// TIA Portal project "MEC10112tHiL2019" (V15)

(* hardware
DEVICE "S7-1200 station_1"  S7-1200 Station
   slot 0: "Rack_0"  S7-1200 Rack  Rack  V1.0
   slot 1: "Simulated Plant Process"  CPU 1214C DC/DC/DC  6ES7 214-1AG40-0XB0  V4.2
      slot 3: "AQ 1x12BIT_1"  AQ1 signal board  6ES7 232-4HA30-0XB0  V1.0
DEVICE "HMI_1"  KTP700 Basic PN
   slot 0: "HMI_1"  KTP700 Basic PN  6AV2 123-2GB03-0AX0  15.0.0.0
   slot 1: "HMI_RT_1"  KTP700 Basic PN  6AV2 123-2GB03-0AX0  15.0.0.0
   slot 5: "HMI_1.IE_CP_1"  PROFINET Interface  15.0.0.0
      slot 1: "PROFINET Interface_1"  PROFINET Interface
         slot 1: "Port_1"  Port
DEVICE "S7-1200 station_2"  S7-1200 Station
   slot 0: "Rack_0"  S7-1200 Rack  Rack  V1.0
   slot 1: "Control Panel PLC"  CPU 1214C AC/DC/Rly  6ES7 214-1BG31-0XB0  V3.0
   slot 3: "AQ 1x12BIT_1"  AQ1 signal board  6ES7 232-4HA30-0XB0  V1.0
DEVICE "SCADA_Display"  SIMATIC PC station
   slot 0: "SIMATIC PC station"  Rail  SIMATIC PC-Station  V1.0
      slot 125: "Stationmanager"  Station_Manager  V6.0.4
   slot 1: "HMI_RT_2"  WinCC RT Advanced  6AV2 104-0xxxx-xxxx  15.0.0.0
      slot 33792: "Host interface"  Host interface
   slot 2: "IE general_1"  IE General  IE_CP  V8.2.0
*)

// ===== PLC "Simulated Plant Process"  CPU 1214C DC/DC/DC =====

VAR_GLOBAL   // PLC tag table "Default tag table"
   "Level" AT %QW80 : Int;
   "OpenV101" AT %I0.0 : Bool;
   "OpenV102" AT %I0.1 : Bool;
   "OpenV103" AT %I0.2 : Bool;
   "OpenV104" AT %I0.3 : Bool;
   "V101OpenLSW" AT %Q0.0 : Bool;
   "V101CloseLSW" AT %Q0.1 : Bool;
   "V102OpenLSW" AT %Q0.2 : Bool;
   "V102CloseLSW" AT %Q0.3 : Bool;
   "V103OpenLSW" AT %Q0.4 : Bool;
   "V103CloseLSW" AT %Q0.5 : Bool;
   "V104OpenLSW" AT %Q0.6 : Bool;
   "V104CloseLSW" AT %Q0.7 : Bool;
   "RunMix" AT %I0.4 : Bool;
   "MinimumHeatTankLevel" AT %Q1.0 : Bool;   // Liquid Level Reached in heating tank
   "MixerRunning" AT %Q1.4 : Bool;
   "Prod_A_Available" AT %Q1.2 : Bool;
   "Prod_B_Available" AT %Q1.3 : Bool;
   "Bottle_Sim_output" AT %Q1.1 : Bool;   // Added output to simulate bottle presence
END_VAR

DATA_BLOCK "TankLevel"   // DB1
{ S7_Optimized_Access := 'FALSE' }
VERSION : 0.1
// stored: InstanceOfName AnalogueOutput_type1
"AnalogueOutput_type1"
BEGIN
END_DATA_BLOCK

DATA_BLOCK "V101"   // DB2
{ S7_Optimized_Access := 'TRUE' }
VERSION : 0.1
// stored: InstanceOfName ValveSim
"ValveSim"
BEGIN
END_DATA_BLOCK

DATA_BLOCK "V102"   // DB3
{ S7_Optimized_Access := 'TRUE' }
VERSION : 0.1
// stored: InstanceOfName ValveSim
"ValveSim"
BEGIN
END_DATA_BLOCK

DATA_BLOCK "V103"   // DB4
{ S7_Optimized_Access := 'TRUE' }
VERSION : 0.1
// stored: InstanceOfName ValveSim
"ValveSim"
BEGIN
END_DATA_BLOCK

DATA_BLOCK "V104"   // DB5
{ S7_Optimized_Access := 'TRUE' }
VERSION : 0.1
// stored: InstanceOfName ValveSim
"ValveSim"
BEGIN
END_DATA_BLOCK

DATA_BLOCK "TankSimulator_DB"   // DB6
{ S7_Optimized_Access := 'TRUE' }
VERSION : 0.1
// stored: InstanceOfName TankSimulator
"TankSimulator"
BEGIN
END_DATA_BLOCK

// folder: System blocks/Program resources

DATA_BLOCK "MixerFB"   // DB7
{ S7_Optimized_Access := 'TRUE' }
AUTHOR : Simatic
FAMILY : IEC
NAME : IEC_TMR
VERSION : 1.0
// stored: InstanceOfName IEC_TIMER
"IEC_TIMER"
BEGIN
END_DATA_BLOCK

// folder: (top level)

FUNCTION_BLOCK "AnalogueInput_type1"   // FB1, SCL
{ S7_Optimized_Access := 'FALSE' }
VERSION : 0.1
   VAR_INPUT
      ChannelAddress : Int;   // PLC Channel Address
      HR : Real := 100.0;   // High Range i.e. Maximum Value of Input Signal
      LR : Real;   // Low Range i.e. Minimum Value of Input Signal
      HSP : Real := 90.0;   // High Alarm Set Point Value
      LSP : Real := 10.0;   // Low Alarm Set Point value
      EnableHSP : Bool := true;   // Enable High Alarm
      EnableLSP : Bool := true;   // Enable Low Alarm
   END_VAR
   VAR_OUTPUT
      PV : Real;   // Process Variable (Scaled Value)
      HighAlarm : Bool;   // High Alarm HSP exceeded
      LowAlarm : Bool;   // Low Alarm LSP exceeded
      HighRangeError : Bool;   // A/D value Exceeds 27,648
      LowRangeError : Bool;   // A/D value lower than 0
   END_VAR
BEGIN
   //This Function Block reads in a value from an anaolgue input channel and
   //scales it between high range (HR) and a low range (LR) values.
   //It also sets high and low value alarms against high (HSP) and low (LSP) set points
   //If the value from the A/D converter exceeds either 0 or 27648 it also generates
   //range error bits

   #PV := ((INT_TO_REAL (#ChannelAddress)*(#HR - #LR))/ 27648.0) + #LR; // Read and scale A/D Value
   IF #EnableHSP=1 THEN                                                 // If High Alarm Enabled
       IF #PV > #HSP THEN                                               // Drive High Alarm
           #HighAlarm := 1;// Statement section IF
       ELSIF #PV< #HSP THEN
           #HighAlarm := 0;
       END_IF;  // Statement section IF
   END_IF;

   IF #EnableLSP=1 THEN                                               // If Low Alarm Enabled
       IF #PV< #LSP THEN                                              // Drive Low Alarm
           #LowAlarm := 1;// Statement section IF
       ELSIF #PV > #LSP THEN
           #LowAlarm := 0;
       END_IF;// Statement section IF
       ;
   END_IF;

   IF #ChannelAddress > 27648 THEN                                 // If A/D value Exceeds 27648
       #HighRangeError := 1;                                       //Out of high range error
       #PV := #HR;                                                 // Limit Output to maximum Value
   END_IF;
   IF #ChannelAddress < 0 THEN                                     // If A/D value is less than 0
       #LowRangeError := 1;                                        // Out of low range error
       #PV := #LR;                                                 // Limit Output to minimum value
   END_IF;
   IF (#ChannelAddress > 0) AND (#ChannelAddress < 27649) THEN     // if in range reset range errors
       #HighRangeError := 0;
       #LowRangeError := 0;
   END_IF;

   //Revision History
   //Tested 25/01/2016
   //Rev 1.0 Added range clipping and error bits
END_FUNCTION_BLOCK

FUNCTION_BLOCK "ValveSim"   // FB2, SCL
{ S7_Optimized_Access := 'TRUE' }
VERSION : 0.1
   VAR_INPUT
      OpenCMD : Bool;
      FaultEnable : Bool;
      OpTime : Int := 20;   // 100ms Increments
   END_VAR
   VAR_OUTPUT
      LimitOpenLSW : Bool;
      LimitCloseLSW : Bool;
   END_VAR
   VAR
      OpenTimer : DInt;
      CloseTimer : DInt;
   END_VAR
BEGIN
   // Valve Open Simulation
   IF #OpenCMD=1 THEN                      //Open CMD
       #OpenTimer := #OpenTimer + 1;       //Inrement Timer
       IF #OpenTimer>=#OpTime AND NOT #FaultEnable THEN   //If Timed value equals or exceeds operaton time
           #LimitOpenLSW := 1;             // Set Limit Switch Feedback
           #OpenTimer:=#OpTime;            // Limit Timer
       END_IF;
   ELSIF #OpenCMD=0 THEN                   // on Close command
       #OpenTimer := 0;                    // Reset Timer
       #LimitOpenLSW := 0;                 // Reset Limit Switch Feedback
   END_IF;

   // Valve Close Simulation
   IF #OpenCMD = 0 THEN                      //Close CMD
       #CloseTimer := #CloseTimer + 1;       //Inrement Timer
       IF #CloseTimer >= #OpTime THEN        //If Timed value equals or exceeds operaton time
           #LimitCloseLSW := 1;              // Set Limit Switch Feedback
           #CloseTimer := #OpTime;           // Limit Timer
       END_IF;
   ELSIF #OpenCMD = 1 THEN                  // on Open command
       #CloseTimer := 0;                    // Reset Timer
       #LimitCloseLSW := 0;                 // Reset Limit Switch Feedback
   END_IF;
END_FUNCTION_BLOCK

FUNCTION_BLOCK "TankSimulator"   // FB3, SCL
{ S7_Optimized_Access := 'TRUE' }
VERSION : 0.1
   VAR_INPUT
      InputValveA : Bool;
      InputValveB : Bool;
      OuputValve : Bool;
      DumpValve : Bool;
      RateA : Real := 0.1;   // litres per 0.1 s
      RateB : Real := 0.1;   // litres per 0.1 s
      RateOut : Real := 0.2;
      HeatLvl_SP : Real := 20.0;
      HR : Real := 110.0;
      LR : Real;
   END_VAR
   VAR_OUTPUT
      "Heat Level" : Bool;
      Level : Real;
   END_VAR
   VAR
      Delta : Real;   // Combined Level Increment
      SimLevel : Real;
   END_VAR
BEGIN
   // Mixing Tank Level Simulator
   // Called from Time Interupt 100mS
   // 
   // Level Change Calculation
   #Delta := 0;                // Reset Delta Change
   IF #InputValveA=1 THEN      // If input valve A open add its rate to Delta
       #Delta:=#Delta + #RateA;
   END_IF;
   IF #InputValveB=1 THEN      // If input valve B open add its rate to Delta
       #Delta := #Delta + #RateB;   
   END_IF;
   IF #OuputValve=1 THEN       // If Output valve open subtract its rate to Delta
       #Delta := #Delta - #RateOut;
   END_IF;
   IF #DumpValve=1 THEN    // If dump valve open level =0
       #Delta := 0;
       #SimLevel := 0;
   END_IF;

   #SimLevel := #SimLevel + #Delta;  // Level Summation
   IF #SimLevel>#HR THEN       // Limit Maximum Level
       #SimLevel := #HR;
   END_IF;
   IF #SimLevel<#LR THEN       // Limit Minimum Level
       #SimLevel := #LR;
   END_IF;

   // Level Above Heat Element
   IF #SimLevel>#HeatLvl_SP THEN // If level covers heating element
       #"Heat Level" := 1;
   ELSIF #SimLevel<#HeatLvl_SP THEN
       #"Heat Level" := 0;
   END_IF;

   // Output Level Simulation
   #Level := #SimLevel;
END_FUNCTION_BLOCK

FUNCTION_BLOCK "AnalogueOutput_type1"   // FB4, SCL
{ S7_Optimized_Access := 'FALSE' }
VERSION : 0.1
   VAR_INPUT
      OP : Real;   // Value to be output to D/A
      HR : Real := 100.0;   // Maximum Value of Output
      LR : Real;   // Minimum Value of Output
   END_VAR
   VAR_OUTPUT
      "Channel Address" : Int;   // D/A Channel Address
      HRexceeded : Bool;   // Input Signal Out of Upper Range
      LRexceeded : Bool;   // Input Signal Out of Lower Range
   END_VAR
BEGIN
   // Function Scales a Real Analogue Value to an integer
   // between 0 and 27648 for driving analogue output card
   // 
   IF (#LR < #OP) AND (#OP < #HR) THEN //If value within range reset error bits
       #HRexceeded := 0;
       #LRexceeded := 0;
   END_IF;
   //
   // Range Real Value
   #"Channel Address":= DINT_TO_INT(ROUND_DINT((#OP*27648.0)/(#HR-#LR)));
   //
   //Range Checking
   IF #OP > #HR THEN                   //Has value exceeded maximum value
       #"Channel Address" := 27648;    //Setoutput to maximum
       #HRexceeded := 1;               //Set error bit
   END_IF;
   IF #OP < #LR THEN                   //Has value exceeded minimum value
       #"Channel Address" := 0;        //Set output to minimum
       #LRexceeded := 1;               //Set error bit
   END_IF;

   //
   //Revision History
   //Rev 1.0 Added range clipping and range errors JMcW 26/01/2016
END_FUNCTION_BLOCK

ORGANIZATION_BLOCK "Main"   // OB1, LAD, ProgramCycle
TITLE = "Main Program Sweep (Cycle)"
{ S7_Optimized_Access := 'TRUE' }
VERSION : 0.1
   VAR_INPUT
      Initial_Call : Bool;   // Initial call of this OB
      Remanence : Bool;   // =True, if remanent data are available
   END_VAR
BEGIN

REGION Network 1: Simulated Tank Level Output Driver
   // Takes simulated value and creates a 0-10v analgue output
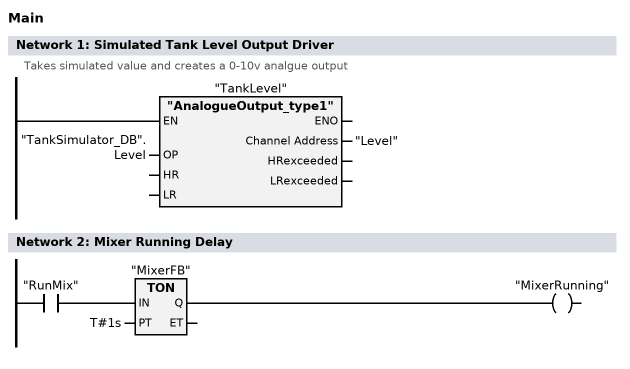
   RUNG wire#powerrail
      "TankLevel"(OP := "TankSimulator_DB".Level, HR :=, LR :=, "Channel Address" => "Level", HRexceeded =>, LRexceeded =>)
   END_RUNG
   // the same network as SCL:
   "TankLevel"(OP := "TankSimulator_DB".Level, "Channel Address" => "Level");   // "AnalogueOutput_type1"
END_REGION

REGION Network 2: Mixer Running Delay
   "MixerFB".TON(IN := "RunMix", PT := T#1s);
   "MixerRunning" := "MixerFB".Q;
END_REGION
END_ORGANIZATION_BLOCK

ORGANIZATION_BLOCK "Cyclic interrupt"   // OB30, LAD, CyclicInterrupt
TITLE = 100mS Cyclic Interupt
{ S7_Optimized_Access := 'TRUE' }
VERSION : 0.1
   VAR_INPUT
      Initial_Call : Bool;   // Initial call of this OB
      Event_Count : Int;   // Events discarded
   END_VAR
BEGIN

REGION Network 1: Inlet Valve 1 Simulation
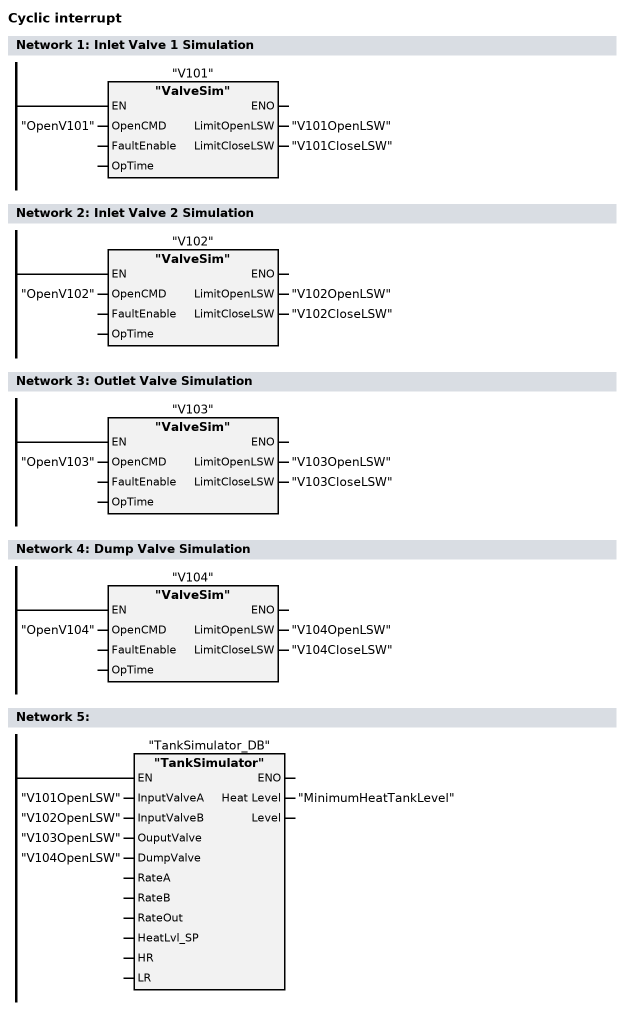
   RUNG wire#powerrail
      "V101"(OpenCMD := "OpenV101", FaultEnable :=, OpTime :=, LimitOpenLSW => "V101OpenLSW", LimitCloseLSW => "V101CloseLSW")
   END_RUNG
   // the same network as SCL:
   "V101"(OpenCMD := "OpenV101", LimitOpenLSW => "V101OpenLSW", LimitCloseLSW => "V101CloseLSW");   // "ValveSim"
END_REGION

REGION Network 2: Inlet Valve 2 Simulation
   RUNG wire#powerrail
      "V102"(OpenCMD := "OpenV102", FaultEnable :=, OpTime :=, LimitOpenLSW => "V102OpenLSW", LimitCloseLSW => "V102CloseLSW")
   END_RUNG
   // the same network as SCL:
   "V102"(OpenCMD := "OpenV102", LimitOpenLSW => "V102OpenLSW", LimitCloseLSW => "V102CloseLSW");   // "ValveSim"
END_REGION

REGION Network 3: Outlet Valve Simulation
   RUNG wire#powerrail
      "V103"(OpenCMD := "OpenV103", FaultEnable :=, OpTime :=, LimitOpenLSW => "V103OpenLSW", LimitCloseLSW => "V103CloseLSW")
   END_RUNG
   // the same network as SCL:
   "V103"(OpenCMD := "OpenV103", LimitOpenLSW => "V103OpenLSW", LimitCloseLSW => "V103CloseLSW");   // "ValveSim"
END_REGION

REGION Network 4: Dump Valve Simulation
   RUNG wire#powerrail
      "V104"(OpenCMD := "OpenV104", FaultEnable :=, OpTime :=, LimitOpenLSW => "V104OpenLSW", LimitCloseLSW => "V104CloseLSW")
   END_RUNG
   // the same network as SCL:
   "V104"(OpenCMD := "OpenV104", LimitOpenLSW => "V104OpenLSW", LimitCloseLSW => "V104CloseLSW");   // "ValveSim"
END_REGION

REGION Network 5
   RUNG wire#powerrail
      "TankSimulator_DB"(InputValveA := "V101OpenLSW", InputValveB := "V102OpenLSW", OuputValve := "V103OpenLSW", DumpValve := "V104OpenLSW", RateA :=, RateB :=, RateOut :=, HeatLvl_SP :=, HR :=, LR :=, "Heat Level" => "MinimumHeatTankLevel", Level =>)
   END_RUNG
   // the same network as SCL:
   "TankSimulator_DB"(InputValveA := "V101OpenLSW",   // "TankSimulator"
                      InputValveB := "V102OpenLSW",
                      OuputValve := "V103OpenLSW",
                      DumpValve := "V104OpenLSW",
                      "Heat Level" => "MinimumHeatTankLevel");
END_REGION
END_ORGANIZATION_BLOCK

// ===== PLC "Control Panel PLC"  CPU 1214C AC/DC/Rly =====

VAR_GLOBAL   // PLC tag table "Default tag table"
   "V101_Opn" AT %I0.0 : Bool;   // Valve 101 Sensor (R101) - Open (NO)
   "V101_Clsd" AT %I0.1 : Bool;   // Valve 101 Sensor (RX101) - Closed (NO)
   "V102_Opn" AT %I0.2 : Bool;   // Valve 102 Sensor (R102)- Open (NO)
   "V102_Clsd" AT %I0.3 : Bool;   // Valve 102 Sensor (RX102)- Closed (NO)
   "V103_Opn" AT %I0.4 : Bool;   // Valve 103 Sensor (R103) - Open (NO)
   "V103_Clsd" AT %I0.5 : Bool;   // Valve 103 Sensor (RX103)- Closed (NO)
   "V104_Opn" AT %I0.6 : Bool;   // Valve 104 Sensor (R104)- Open (NO)
   "V104_Clsd" AT %I0.7 : Bool;   // Valve 104 Sensor (RX104)- Clsd (NO)
   "ProdA_level_OK" AT %I1.0 : Bool;   // ProdA (RXOrange) - Clsd (NO)
   "ProdB_level_OK" AT %I1.1 : Bool;   // ProdB (RXGreen) - Clsd (NO)
   "Bottle_Pos_OK" AT %I1.2 : Bool;   // Bottle (RXPurple) - Clsd (NO)
   "Mixer_Detect_On" AT %I1.3 : Bool;   // Mixer Detected ON (RXBlue) - Clsd (KM1- NO)
   "Temp_Mixer_Analog" AT %IW64 : Int;   // Temperature Measurement (AT) - Analogue Input
   "Liquid_Level_Analog" AT %IW66 : Int;   // Liquid Level Measurement in Tank (AS) - Analogue Input
   "EMS" AT %I1.5 : Bool;   // EMS Push Button (+ES+) - Open (NC)
   "Liquid_Level_ProcTank_Min" AT %I1.4 : Bool;   // Processing Tank Minimum Level (RXGrey) - Closed (NO)
   "V101_On" AT %Q0.0 : Bool;   // V101 Valve (S101) - ON (NO)
   "V102_On" AT %Q0.1 : Bool;   // V102 Valve (S102) - ON (NO)
   "V103_On" AT %Q0.2 : Bool;   // V103 Valve (S103) - ON (NO)
   "V104_On" AT %Q0.3 : Bool;   // V104 Valve (S104) - ON (NO)
   "Mixer_On" AT %Q0.4 : Bool;   // Mixer On (Y+1) - ON (KM1 Contactor)
   "Heater_On" AT %Q0.5 : Bool;   // Heater On (Y+2) - ON (NO)
   "Fan_On" AT %Q0.6 : Bool;   // Fan On (Y+3) - ON (NO)
   "Conveyor_On" AT %Q1.0 : Bool;   // Conveyor On (Y+4) - ON (NO)
   "Reverse_On" AT %Q1.1 : Bool;   // Conveyor Set to Reverse (Y+5) - ON (NO)
   "Conveyor_Speed" AT %QW80 : Int;   // Conveyor Speed Control (SY+) - Analogue Output
   "Start_PB" AT %M10.0 : Bool;   // Start Machine Push Button (HMI) - NO
   "Stop_PB" AT %M11.0 : Bool;   // Stop Process Push Button (HMI) - NO
   "Auto_Mode" AT %M12.0 : Bool;   // Automatic Mode Selected (HMI) - NO
   "Manual_Mode" AT %M13.0 : Bool;   // Manual Mode Selected (HMI) - NO
   "Forced_Manual_Mode" AT %M14.0 : Bool;   // Forced Manual Mode Engaged - NO
   "Reset_PB" AT %M15.0 : Bool;   // Reset Process Push Button (HMI) - NO
   "ProdA_SP_Rec1" AT %MW100 : Int;   // Recipe 1 Product A Set point in Litres - Int
   "ProdB_SP_Rec1" AT %MW102 : Int;   // Recipe 1 Product B Set point in Litres - Int
   "ProdA_Tol_Rec1" AT %MW104 : Int;   // Recipe 1 Product A Tolerance in Litres - Int
   "ProdB_Tol_Rec1" AT %MW106 : Int;   // Recipe 1 Product B Tolerance in Litres - Int
   "Mix_Temp_SP_Rec1" AT %MW108 : Int;   // Recipe 1 Mix Temperature Setpoint in degree C- Int
   "Mix_Temp_Tol_Rec1" AT %MW110 : Int;   // Recipe 1 Mix Temperature Tolerance in degree C- Int
   "Mix_Time_Rec1" AT %MW112 : Int;   // Recipe 1 Mixing Time in Milliseconds - Int
   "Bottle_Size_Rec1" AT %MW114 : Int;   // Recipe 1 Bottle Size in Litres - Int
   "Bottle_Batch_Size_Rec1" AT %MW116 : Int;   // Recipe 1 Number of Bottles required - Int
   "Recipe_1" AT %M118.0 : Bool;   // Set Recipe 1 Selection Button
   "Recipe_2" AT %M119.0 : Bool;   // Set Recipe 2 Selection Button
   "Recipe_3" AT %M120.0 : Bool;   // Set Recipe 3 Selection Button
   "ProdA_SP_Rec2" AT %MW200 : Int;   // Recipe 2 Product A Set point in Litres - Int
   "ProdB_SP_Rec2" AT %MW122 : Int;   // Recipe 2 Product B Set point in Litres - Int
   "ProdA_Tol_Rec2" AT %MW124 : Int;   // Recipe 2 Product A Tolerance in Litres - Int
   "ProdB_Tol_Rec2" AT %MW126 : Int;   // Recipe 2 Product B Tolerance in Litres - Int
   "Mix_Temp_SP_Rec2" AT %MW128 : Int;   // Recipe 2 Mix Temperature Setpoint in degree C- Int
   "Mix_Temp_Tol_Rec2" AT %MW130 : Int;   // Recipe 2 Mix Temperature Tolerance in degree C- Int
   "Mix_Time_Rec2" AT %MW132 : Int;   // Recipe 2 Mixing Time in Milliseconds - Int
   "Bottle_Size_Rec2" AT %MW134 : Int;   // Recipe 2 Bottle Size in Litres - Int
   "Bottle_Batch_Size_Rec2" AT %MW136 : Int;   // Recipe 2 Number of Bottles required - Int
   "ProdA_SP_Rec3" AT %MW138 : Int;   // Recipe 3 Product A Set point in Litres - Int
   "ProdB_SP_Rec3" AT %MW140 : Int;   // Recipe 3 Product B Set point in Litres - Int
   "ProdA_Tol_Rec3" AT %MW142 : Int;   // Recipe 3 Product A Tolerance in Litres - Int
   "ProdB_Tol_Rec3" AT %MW144 : Int;   // Recipe 3 Product B Tolerance in Litres - Int
   "Mix_Temp_SP_Rec3" AT %MW146 : Int;   // Recipe 3 Mix Temperature Setpoint in degree C- Int
   "Mix_Temp_Tol_Rec3" AT %MW148 : Int;   // Recipe 3 Mix Temperature Tolerance in degree C- Int
   "Mix_Time_Rec3" AT %MW150 : Int;   // Recipe 3 Mixing Time in Milliseconds - Int
   "Bottle_Size_Rec3" AT %MW152 : Int;   // Recipe 3 Bottle Size in Litres - Int
   "Bottle_Batch_Size_Rec3" AT %MW154 : Int;   // Recipe 3 Number of Bottles required - Int
   "Error_Status" AT %M404.0 : Bool;   // Error Status Bit
   "Analog_Level" AT %MW160 : Int;   // Analog Level memory location
   "Step_1" AT %M50.0 : Bool;   // System Sequence Step 1 - Automatic Enabled
   "Step_2" AT %M51.0 : Bool;   // System Sequence Step 2 - Product A being filled
   "Step_3" AT %M52.0 : Bool;   // System Sequence Step 3 - Product B being filled
   "Step_4" AT %M53.0 : Bool;   // System Sequence Step 4 - Mixer and Heating On
   "Step_5" AT %M54.0 : Bool;   // System Sequence Step 5 - Cooking process
   "Step_6" AT %M55.0 : Bool;   // System Sequence Step 6 - Start bottle Filling Process (conveyor ON)
   "Step_7" AT %M56.0 : Bool;   // System Sequence Step 7 - Fill the bottle.
   "Step_8" AT %M60.0 : Bool;   // System Sequence Step 8 - Bottle filled.
   "Step_9" AT %M58.0 : Bool;   // System Sequence Step 9 - Reset filling loop/Reset batch.
   "Temp_in_Range" AT %M600.0 : Bool;   // Temperature of Heater is within Range
   "Mixing_done" AT %M61.0 : Bool;   // Mixing process complete
   "Bottle_Count" AT %MW156 : Int;   // Bottle Count Number (memory bit)
   "System_Enabled" AT %M164.0 : Bool;   // System On (memory bit)
   "Conveyor_Speed_value" AT %MD300 : Real;   // Speed value input (memory bit)
   "End_cycle" AT %M165.0 : Bool;   // End of batch
   "V101_Man" AT %M165.1 : Bool;   // V101 Manual Activation
   "V102_Man" AT %M165.2 : Bool;   // V102 Manual Activation
   "V103_Man" AT %M165.3 : Bool;   // V103 Manual Activation
   "V104_Man" AT %M165.4 : Bool;   // V104 Manual Activation
   "Heating_Man" AT %M165.5 : Bool;   // Heating Manual Activation
   "Conveyor_Man" AT %M165.6 : Bool;   // Conveyor Manual Activation
   "Valve_Error" AT %M165.7 : Bool;   // Valve Error Tag
   "Heater_liquid_error" AT %M166.0 : Bool;   // Heater liquid level Error Tag
   "Conveyor_error" AT %M166.1 : Bool;   // Conveyor Error Tag
   "ProdA_Level_Error" AT %M166.2 : Bool;   // Product A Tank Empty
   "ProdB_Level_Error" AT %M166.3 : Bool;   // Product B Tank Empty
   "Liquid_Error" AT %M166.4 : Bool;   // Main Liquid Error
   "Overflow_Error" AT %M166.5 : Bool;   // Main Tank Overflow Error
   "EMS_Triggered" AT %M166.6 : Bool;   // EMS
END_VAR

DATA_BLOCK "Ultrasonic_Lvl_In_DB"   // DB1
{ S7_Optimized_Access := 'TRUE' }
VERSION : 0.1
// stored: InstanceOfName Analog_In
"Analog_In"
BEGIN
END_DATA_BLOCK

DATA_BLOCK "Purging_Valve(V104)_DB"   // DB2
{ S7_Optimized_Access := 'TRUE' }
VERSION : 0.1
// stored: InstanceOfName Valve
"Valve"
BEGIN
END_DATA_BLOCK

DATA_BLOCK "System_Mode_Selection_DB"   // DB3
{ S7_Optimized_Access := 'TRUE' }
VERSION : 0.1
// stored: InstanceOfName RunMode_Selection
"RunMode_Selection"
BEGIN
END_DATA_BLOCK

DATA_BLOCK "Low_Pass_Filter_DB"   // DB4
{ S7_Optimized_Access := 'TRUE' }
VERSION : 0.1
// stored: InstanceOfName Low_Pass_Filter
"Low_Pass_Filter"
BEGIN
END_DATA_BLOCK

DATA_BLOCK "Recipe Selection_DB"   // DB5
{ S7_Optimized_Access := 'TRUE' }
VERSION : 0.1
// stored: InstanceOfName Recipe Selection
"Recipe Selection"
BEGIN
END_DATA_BLOCK

DATA_BLOCK "Valve_ProdB(V102)"   // DB7
{ S7_Optimized_Access := 'TRUE' }
VERSION : 0.1
// stored: InstanceOfName Valve
"Valve"
BEGIN
END_DATA_BLOCK

DATA_BLOCK "Filling Control_DB"   // DB8
{ S7_Optimized_Access := 'TRUE' }
VERSION : 0.1
// stored: InstanceOfName Filling Control
"Filling Control"
BEGIN
END_DATA_BLOCK

DATA_BLOCK "Temperature_Measurement_In"   // DB10
{ S7_Optimized_Access := 'TRUE' }
VERSION : 0.1
// stored: InstanceOfName Analog_In
"Analog_In"
BEGIN
END_DATA_BLOCK

DATA_BLOCK "Analogue Output_Conveyor_Speed"   // DB12
{ S7_Optimized_Access := 'TRUE' }
VERSION : 0.1
// stored: InstanceOfName Analogue Output
"Analogue Output"
BEGIN
END_DATA_BLOCK

DATA_BLOCK "Valve_Bottle_Fill(V103)"   // DB13
{ S7_Optimized_Access := 'TRUE' }
VERSION : 0.1
// stored: InstanceOfName Valve
"Valve"
BEGIN
END_DATA_BLOCK

DATA_BLOCK "Valve_ProdA(V101)"   // DB14
{ S7_Optimized_Access := 'TRUE' }
VERSION : 0.1
// stored: InstanceOfName Valve
"Valve"
BEGIN
END_DATA_BLOCK

DATA_BLOCK "Error_Tolerance_ProductAandB"   // DB17
{ S7_Optimized_Access := 'TRUE' }
VERSION : 0.1
// stored: InstanceOfName Error_Tolerance
"Error_Tolerance"
BEGIN
END_DATA_BLOCK

// folder: System blocks/Program resources

DATA_BLOCK "Delay_Timer"   // DB9
{ S7_Optimized_Access := 'TRUE' }
AUTHOR : Simatic
FAMILY : IEC
NAME : IEC_TMR
VERSION : 1.0
// stored: InstanceOfName IEC_TIMER
"IEC_TIMER"
BEGIN
END_DATA_BLOCK

DATA_BLOCK "Mixing_Timer"   // DB11
{ S7_Optimized_Access := 'TRUE' }
AUTHOR : Simatic
FAMILY : IEC
NAME : IEC_TMR
VERSION : 1.0
// stored: InstanceOfName IEC_TIMER
"IEC_TIMER"
BEGIN
END_DATA_BLOCK

DATA_BLOCK "Bottle_Produced_UP"   // DB15
{ S7_Optimized_Access := 'TRUE' }
AUTHOR : Simatic
FAMILY : IEC
NAME : CNTR
VERSION : 1.0
// stored: InstanceOfName IEC_COUNTER
"IEC_COUNTER"
BEGIN
END_DATA_BLOCK

DATA_BLOCK "Purge_Timer"   // DB16
{ S7_Optimized_Access := 'TRUE' }
AUTHOR : Simatic
FAMILY : IEC
NAME : IEC_TMR
VERSION : 1.0
// stored: InstanceOfName IEC_TIMER
"IEC_TIMER"
BEGIN
END_DATA_BLOCK

DATA_BLOCK "Timer_Conveyor"   // DB19
{ S7_Optimized_Access := 'TRUE' }
AUTHOR : Simatic
FAMILY : IEC
NAME : IEC_TMR
VERSION : 1.0
// stored: InstanceOfName IEC_TIMER
"IEC_TIMER"
BEGIN
END_DATA_BLOCK

// folder: (top level)

FUNCTION_BLOCK "RunMode_Selection"   // FB1, SCL
{ S7_Optimized_Access := 'TRUE' }
VERSION : 0.1
   VAR_INPUT
      Fault : Bool;   // Fault detected
      AutoMan_Selec : Bool;   // Auto Mode Selected
   END_VAR
   VAR_OUTPUT
      Forced_Manual : Bool;   // Forced Manual Mode Confirmed
      Manual : Bool;   // Manual Mode Confirmed
      Automatic : Bool;   // Automatic Mode Confirmed
   END_VAR
   VAR RETAIN
      state : Int := 1;
   END_VAR
BEGIN
   // The function creates an interlock between the various run mode of the process.
   CASE #state OF
       1: //Forced Manual State.
           IF (#AutoMan_Selec = 0 AND #Fault = 0) THEN
               #state := 2; // Manual Mode Validated.
           END_IF;
           IF (#AutoMan_Selec = 1 AND #Fault = 0) THEN
               #state := 3; //Automatic Mode Validated.
           END_IF;
           #Forced_Manual := 1; //Machine Mode Outputs.
           #Manual := 0;
           #Automatic := 0;
       2: //Manual State.
           IF #Fault = 1 THEN
               #state := 1; //Forced Manual Validated.
           END_IF;
           IF (#AutoMan_Selec = 1 AND #Fault = 0) THEN
               #state := 3; //Automatic Mode Validated.
           END_IF;
           #Forced_Manual := 0; //Machine Mode Outputs.
           #Manual := 1;
           #Automatic := 0;
       3: //Automatic State.
           IF #Fault = 1 THEN
               #state := 1; //Force Manual Validated.
           END_IF;
           IF (#AutoMan_Selec = 0 AND #Fault = 0) THEN
               #state := 2; //Manual Mode Validated
           END_IF;
           #Forced_Manual := 0; //Machine Mode Outputs
           #Manual := 0;
           #Automatic := 1;
   END_CASE;
END_FUNCTION_BLOCK

FUNCTION_BLOCK "Low_Pass_Filter"   // FB3, SCL
{ S7_Optimized_Access := 'TRUE' }
VERSION : 0.1
   VAR_INPUT
      Xf : Real;   // Input to filter
      Tc : Real := 2.0;   // Time Constant in seconds (default 2.0s)
      Ts : Real := 0.1;   // Sample Time (default 100ms)
   END_VAR
   VAR_OUTPUT
      Output : Int;
   END_VAR
   VAR_IN_OUT
      Yn_1 : Real;   // Previous Filter Output Value
      Kf : Real;   // Filter Gain = Ts/(Ts+Tc)
      Yf : Real;   // Filter output
   END_VAR
BEGIN
   // This function block is low pass filter.
   // The filter blocks higher frequency to allow a smoother signal.

   //Filter Constant.
   #Kf := #Ts / (#Ts + #Tc);
   //Filter Output.
   #Yf := #Yn_1 + (#Kf * (#Xf - #Yn_1));
   #Yn_1 := #Yf;
   #Output := REAL_TO_INT(#Yn_1);
END_FUNCTION_BLOCK

FUNCTION_BLOCK "Valve"   // FB4, SCL
{ S7_Optimized_Access := 'TRUE' }
VERSION : 0.1
   VAR_INPUT
      Valve_Sens_Open : Bool;   // Valve Sensor State: Open
      "Valve_ Sens_ Closed" : Bool;   // Valve Sensor State: Closed
      Level_Ok : Bool;   // Tank Sensor: Level OK
      Valve_Opn_Req : Bool;   // Valve Open Request Input
      Manual_mode : Bool;   // Manual Mode requested
   END_VAR
   VAR_OUTPUT
      Valve_Control : Bool;   // Valve Control. (True=Open ; False=Close)
      Valve_Error : Bool;   // Valve Error Status
   END_VAR
   VAR
      OpenTimer : DInt;
      CloseTimer : DInt;
   END_VAR
BEGIN
   // Valve Control and Error Management Function
   // If Valve is Requested and no error:
   IF #Valve_Opn_Req = 1 AND #Valve_Error=0 THEN
       //Turn OpenTimer ON and Reset Closetimer
       #OpenTimer := #OpenTimer + 1;
       #CloseTimer := 0;
       //If Valve_Control is OFF and Timer>=3 then Valve Error.
       IF #Valve_Control = 0 AND #OpenTimer >= 3 THEN
           #Valve_Error := 1;
           //If Sensors and Level Ok then Output ok.
       ELSIF #Level_Ok = 1 THEN
           #Valve_Control := 1;
       END_IF;
   END_IF;

   //If Valve off requested and no error: 
   IF #Valve_Opn_Req = 0 AND #Valve_Error = 0 THEN
       //Reset OpenTimer and Start CloseTimer.
       #CloseTimer := #CloseTimer + 1;
       #OpenTimer := 0;
       //If Valve_Control is ON and CloseTimer>=3 then valve error
       IF #Valve_Control = 1 AND #CloseTimer >= 3 THEN
           #Valve_Error := 1;
       //Else Close Valve
       ELSE
           #Valve_Control := 0;
       END_IF;
   END_IF;
   //Sensor Error: If Sensors both open or both closed then error
    IF #Valve_Sens_Open = 0 AND #"Valve_ Sens_ Closed" = 0 OR #Valve_Sens_Open = 1 AND #"Valve_ Sens_ Closed" = 1 THEN
        #Valve_Error := 1;
    ELSIF #Valve_Sens_Open = 0 AND #"Valve_ Sens_ Closed" = 1 OR #Valve_Sens_Open = 1 AND #"Valve_ Sens_ Closed" = 0 THEN
        #Valve_Error := 0;
    END_IF;
    //If Manual Mode is engaged and valve is on then valve error is overriden.
    IF #Manual_mode = 1 AND #Valve_Control = 1 THEN
        #Valve_Error := 0;
    END_IF;
END_FUNCTION_BLOCK

FUNCTION_BLOCK "Recipe Selection"   // FB5, SCL
{ S7_Optimized_Access := 'TRUE' }
VERSION : 0.1
   VAR_INPUT
      Bottle_Size_Rec1 : Int;   // Parameter Input Rec 1
      Bottle_Number_Rec1 : Int;   // Parameter Input Rec 1
      Product_A_Rec1 : Int;   // Parameter Input Rec 1
      Product_A_Tol_Rec1 : Int;   // Parameter Input Rec 1
      Product_B_Rec1 : Int;   // Parameter Input Rec 1
      Product_B_Tol_Rec1 : Int;   // Parameter Input Rec 1
      Mix_Temp_Rec1 : Int;   // Parameter Input Rec 1
      Mix_Temp_Tol_Rec1 : Int;   // Parameter Input Rec 1
      Mixing_Time_Rec1 : Int;   // Parameter Input Rec 1
      Bottle_Size_Rec2 : Int;   // Parameter Input Rec 2
      Bottle_Number_Rec2 : Int;   // Parameter Input Rec 2
      Product_A_Rec2 : Int;   // Parameter Input Rec 2
      Product_A_Tol_Rec2 : Int;   // Parameter Input Rec 2
      Product_B_Rec2 : Int;   // Parameter Input Rec 2
      Product_B_Tol_Rec2 : Int;   // Parameter Input Rec 2
      Mix_Temp_Rec2 : Int;   // Parameter Input Rec 2
      Mix_Temp_Tol_Rec2 : Int;   // Parameter Input Rec 2
      Mixing_Time_Rec2 : Int;   // Parameter Input Rec 2
      Bottle_Size_Rec3 : Int;   // Parameter Input Rec 3
      Bottle_Number_Rec3 : Int;   // Parameter Input Rec 3
      Product_A_Rec3 : Int;   // Parameter Input Rec 3
      Product_A_Tol_Rec3 : Int;   // Parameter Input Rec 3
      Product_B_Rec3 : Int;   // Parameter Input Rec 3
      Product_B_Tol_Rec3 : Int;   // Parameter Input Rec 3
      Mix_Temp_Rec3 : Int;   // Parameter Input Rec 3
      Mix_Temp_Tol_Rec3 : Int;   // Parameter Input Rec 3
      Mixing_Time_Rec3 : Int;   // Parameter Input Rec 3
      "Recipe 1" : Bool;   // Recipe 1 Selection
      "Recipe 2" : Bool;   // Recipe 2 Selection
      Reset : Bool;   // Reset Function Input
      "Recipe 3" : Bool;   // Recipe 3 Selection
   END_VAR
   VAR_OUTPUT
      Bottle_Size : Int;   // Parameter output
      Bottle_Number : Int;   // Parameter output
      Product_A : Int;   // Parameter output
      Product_A_Tol : Int;   // Parameter output
      Product_B : Int;   // Parameter output
      Product_B_Tol : Int;   // Parameter output
      Mix_Temp : Int;   // Parameter output
      Mix_Temp_Tol : Int;   // Parameter output
      Mixing_Time : DInt;   // Parameter output
      "Batch_Size_A+B" : Int;   // Parameter output
      Recipe_Selected_Out : Bool;   // Recipe Selected
   END_VAR
   VAR RETAIN
      State : Int := 1;   // Case state
   END_VAR
BEGIN
   // This Function allows to create an interlock between different recipes. 
   // The function will input all recipes parameters and output a single set of parameters

   CASE #State OF
       1: //Recipe Selection
           #Recipe_Selected_Out := 0;
           IF (#"Recipe 1" = 1 AND #"Recipe 2" = 0 AND #"Recipe 3" = 0) THEN
               #State := 2; //Recipe 1 parameters passed.
           END_IF;
           IF (#"Recipe 1" = 0 AND #"Recipe 2" = 1 AND #"Recipe 3" = 0) THEN
               #State := 3; //Recipe 2 parameters passed.

           END_IF;
           IF (#"Recipe 1" = 0 AND #"Recipe 2" = 0 AND #"Recipe 3" = 1) THEN
               #State := 4; //Recipe 3 parameters passed.
           END_IF;
       2: //Recipe 1.
           #Bottle_Size := #Bottle_Size_Rec1;
           #Bottle_Number := #Bottle_Number_Rec1;
           #Product_A := #Product_A_Rec1;
           #Product_A_Tol := #Product_A_Tol_Rec1;
           #Product_B := #Product_B_Rec1;
           #Product_B_Tol := #Product_B_Tol_Rec1;
           #Mix_Temp := #Mix_Temp_Rec1;
           #Mix_Temp_Tol := #Mix_Temp_Tol_Rec1;
           #Mixing_Time := #Mixing_Time_Rec1;
           #"Batch_Size_A+B" := #Product_A + #Product_B;
           #Recipe_Selected_Out := 1;
           IF #Reset = 1 THEN
               #State := 1;
           END_IF;
       3: //Recipe 2
           #Bottle_Size := #Bottle_Size_Rec2;
           #Bottle_Number := #Bottle_Number_Rec2;
           #Product_A := #Product_A_Rec2;
           #Product_A_Tol := #Product_A_Tol_Rec2;
           #Product_B := #Product_B_Rec2;
           #Product_B_Tol := #Product_B_Tol_Rec2;
           #Mix_Temp := #Mix_Temp_Rec2;
           #Mix_Temp_Tol := #Mix_Temp_Tol_Rec2;
           #Mixing_Time := #Mixing_Time_Rec2;
           #"Batch_Size_A+B" := #Product_A + #Product_B;
           #Recipe_Selected_Out := 1;
           IF #Reset = 1 THEN
               #State := 1;
           END_IF;
       4: //Recipe 3
           #Bottle_Size := #Bottle_Size_Rec3;
           #Bottle_Number := #Bottle_Number_Rec3;
           #Product_A := #Product_A_Rec3;
           #Product_A_Tol := #Product_A_Tol_Rec3;
           #Product_B := #Product_B_Rec3;
           #Product_B_Tol := #Product_B_Tol_Rec3;
           #Mix_Temp := #Mix_Temp_Rec3;
           #Mix_Temp_Tol := #Mix_Temp_Tol_Rec3;
           #Mixing_Time := #Mixing_Time_Rec3;
           #"Batch_Size_A+B" := #Product_A + #Product_B;
           #Recipe_Selected_Out := 1;
           IF #Reset = 1 THEN
               #State := 1;
           END_IF;

   END_CASE;
END_FUNCTION_BLOCK

FUNCTION_BLOCK "Filling Control"   // FB6, SCL
{ S7_Optimized_Access := 'TRUE' }
VERSION : 0.1
   VAR_INPUT
      Trigger : Bool;
      Level : Real;
      "Unit Size" : Int;
   END_VAR
   VAR_OUTPUT
      Target_Lvl : Real;
   END_VAR
BEGIN
   // Filling Process Control - The Function will calculate the new tank level target 
   // according to to the size per unit for every trigger.

   IF #Trigger = 1 THEN
       #Target_Lvl := #Level;
       #Target_Lvl := #Target_Lvl - #"Unit Size";
   END_IF;
END_FUNCTION_BLOCK

FUNCTION_BLOCK "Analogue Output"   // FB7, SCL
{ S7_Optimized_Access := 'TRUE' }
VERSION : 0.1
   VAR_INPUT
      OP : Real := 0.0;   // Value to be output to D/A
      HR : Real := 4.0;   // Maximum Value of Output
      LR : Real := 8.0;   // Minimum Value of Output
   END_VAR
   VAR_OUTPUT
      "Channel Address" : Int := 0;   // D/A Channel Address
      HRexceeded : Bool := 0;   // Input Signal Out of Upper Range
      LRexceeded : Bool := 0;   // Input Signal Out of Lower Range
   END_VAR
BEGIN
   // Function Scales a Real Analogue Value to an integer
   // Between 0 and 27648 for driving the output card
   IF (#LR < #OP) AND (#OP < #HR) THEN
       #HRexceeded := 0;
       #LRexceeded := 0;
   END_IF;
   //
   // Range Real Value
   #"Channel Address" := DINT_TO_INT(ROUND((#OP * 27648.0) / (#HR - #LR)));
   //
   //Range Checking
   IF #OP > #HR THEN
       #"Channel Address" := 27648;
       #HRexceeded := 1;
   END_IF;
   IF #OP < #LR THEN
       #"Channel Address" := 0;
       #LRexceeded := 1;
   END_IF;
END_FUNCTION_BLOCK

FUNCTION_BLOCK "Analog_In"   // FB8, SCL
{ S7_Optimized_Access := 'TRUE' }
VERSION : 0.1
   VAR_INPUT
      ChannelAddress : Int;
      HR : Real := 100.0;
      LR : Real := -100.0;
      HSP : Real := 90.0;
      LSP : Real := 10.0;
      EnableHSP : Bool := true;
      EnableLSP : Bool := true;
   END_VAR
   VAR_OUTPUT
      PV : Real;
      HighAlarm : Bool;
      LowAlarm : Bool;
      HighRangeError : Bool;
      LowRangeError : Bool;
   END_VAR
BEGIN
   // This function block reads analogue input channel and scales
   // between HR (High Range) and LR (Low Range) values
   // Sets Low and High alarm values against HSP and LSP
   // If the A/D converter values are below 0 or over 27648 an error 
   // will be generated

   #PV := ((INT_TO_REAL(#ChannelAddress) * (#HR - #LR)) / 27648) + #LR; // Read and scale A/D Values
   IF #EnableHSP = 1 THEN                                          // If High Alarm Enabled
       IF #PV > #HSP THEN                                          // Drive High Alarm
           #HighAlarm := 1;
       ELSIF #PV < #HSP THEN
           #HighAlarm := 0;
       END_IF;
   END_IF;

   IF #EnableLSP = 1 THEN                                          // If Low Alarm Enabled
       IF #PV < #LSP THEN                                          // Drive Low Alarm
           #LowAlarm := 1;
       ELSIF #PV > #LSP THEN
           #LowAlarm := 0;
       END_IF;
   END_IF;
   IF #ChannelAddress > 27648 THEN                                 // If A/D Values over 27648
       #HighRangeError := 1;                                       // Out of high limit
       #PV := #HR;                                                 // Limit output to maximum value
   END_IF;
   IF #ChannelAddress < 0 THEN                                     // if A/D Values below 0
       #LowRangeError := 1;                                        // Out of low limit
       #PV := #LR;                                                  // Limit output to minimum value
   END_IF;
   IF (#ChannelAddress > 0) AND (#ChannelAddress < 27648) THEN
       #HighRangeError := 0;
       #LowRangeError := 0;
   END_IF;

   //Revision History
   //Tested
   //REV 1.0
END_FUNCTION_BLOCK

FUNCTION_BLOCK "Error_Tolerance"   // FB9, SCL
{ S7_Optimized_Access := 'TRUE' }
VERSION : 0.1
   VAR_INPUT
      Product_1 : Int;
      Product_2 : Int;
      Prod1_Tolerance : Int;
      Prod2_Tolerance : Int;
      Value_Read : Real;
      Reset : Bool;
   END_VAR
   VAR_OUTPUT
      Error_Output : Bool;
   END_VAR
   VAR
      TimerError : DInt;
   END_VAR
   VAR_TEMP
      Error_level : Bool;
      Temp_Value : Int;
   END_VAR
BEGIN
   // Function manages the tolerance level error between two products.
       //Product 1 Tolerance Level Error Management.
       IF #Value_Read > #Product_1 + #Prod1_Tolerance THEN
           #Temp_Value := #Product_1 + #Prod1_Tolerance;
           #Error_level:=1;
       ELSIF #Value_Read < #Product_1 - #Prod1_Tolerance THEN
           #Temp_Value := #Product_1 + #Prod1_Tolerance;
           #Error_level := 1;
       END_IF;
       //Product 2 Tolerance Level Error Management.
       IF #Value_Read > #Temp_Value + #Product_2 + #Prod2_Tolerance THEN
           #Error_level := 1;
       ELSIF #Value_Read < #Temp_Value + #Product_2 - #Prod2_Tolerance THEN
           #Error_level := 1;
       END_IF;
       //If and Error in the level is triggered the system has 30s to stabilise or reach level
       //IF #Error_level = 1 AND #Reset=0 THEN
        //   #TimerError := #TimerError + 1;
       //    IF #TimerError >= 30 THEN
        //       #Error_Output := 1;
               //If Reset triggered then reset timer.
       //    ELSIF #Reset = 1 OR #Error_level = 0 THEN
       //        #TimerError := 0;
       //    END_IF;
      // END_IF;
END_FUNCTION_BLOCK

FUNCTION "System Process Control" : Void   // FC1, LAD
TITLE = System Process Control.
{ S7_Optimized_Access := 'TRUE' }
VERSION : 0.1
// The Sytem Process Control manages:
// - System Enable (ON/OFF)
// - Process Mode: Automatic, Manual or Forced Manual.
// - Recipe Selection: Recipe 1, Recipe 2 or Recipe 3.
// - Process Sequence.
   VAR_TEMP   // added for the SCL form of the ladder/FBD networks
      _w1 : Bool;
   END_VAR
BEGIN

REGION Network 1: System Enable and Process Mode Selection
   // Creates an interlock between the different run modes of the system.
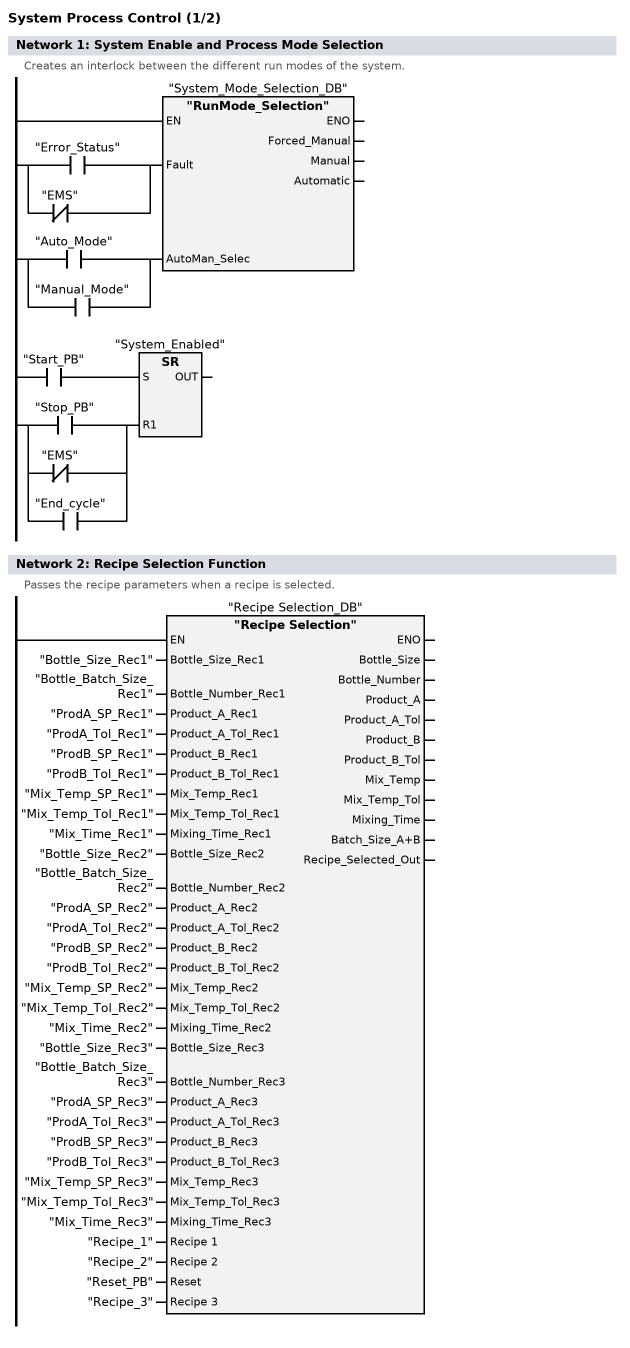
   RUNG wire#powerrail
      "System_Mode_Selection_DB"(Fault := wire#w1, AutoMan_Selec := wire#w2, Forced_Manual =>, Manual =>, Automatic =>)
   END_RUNG
   RUNG wire#powerrail
      Contact( "Error_Status" )
   END_RUNG wire#w1
   RUNG wire#powerrail
      I_Contact( "EMS" )
   END_RUNG wire#w1
   RUNG wire#powerrail
      Contact( "Auto_Mode" )
   END_RUNG wire#w2
   RUNG wire#powerrail
      Contact( "Manual_Mode" )
   END_RUNG wire#w2
   RUNG wire#powerrail
      Contact( "Start_PB" )
      S_SR(operand := "System_Enabled", r1 := wire#w3)
   END_RUNG
   RUNG wire#powerrail
      Contact( "Stop_PB" )
   END_RUNG wire#w3
   RUNG wire#powerrail
      I_Contact( "EMS" )
   END_RUNG wire#w3
   RUNG wire#powerrail
      Contact( "End_cycle" )
   END_RUNG wire#w3
   // the same network as SCL:
   "System_Mode_Selection_DB"(Fault := "Error_Status" OR NOT "EMS",   // "RunMode_Selection"
                           AutoMan_Selec := "Auto_Mode" OR "Manual_Mode");
   IF "Start_PB" THEN
       "System_Enabled" := TRUE;   // SR flip-flop
   END_IF;
   IF "Stop_PB" OR NOT "EMS" OR "End_cycle" THEN "System_Enabled" := FALSE; END_IF;
END_REGION

REGION Network 2: Recipe Selection Function
   // Passes the recipe parameters when a recipe is selected.
   RUNG wire#powerrail
      "Recipe Selection_DB"(Bottle_Size_Rec1 := "Bottle_Size_Rec1", Bottle_Number_Rec1 := "Bottle_Batch_Size_Rec1", Product_A_Rec1 := "ProdA_SP_Rec1", Product_A_Tol_Rec1 := "ProdA_Tol_Rec1", Product_B_Rec1 := "ProdB_SP_Rec1", Product_B_Tol_Rec1 := "ProdB_Tol_Rec1", Mix_Temp_Rec1 := "Mix_Temp_SP_Rec1", Mix_Temp_Tol_Rec1 := "Mix_Temp_Tol_Rec1", Mixing_Time_Rec1 := "Mix_Time_Rec1", Bottle_Size_Rec2 := "Bottle_Size_Rec2", Bottle_Number_Rec2 := "Bottle_Batch_Size_Rec2", Product_A_Rec2 := "ProdA_SP_Rec2", Product_A_Tol_Rec2 := "ProdA_Tol_Rec2", Product_B_Rec2 := "ProdB_SP_Rec2", Product_B_Tol_Rec2 := "ProdB_Tol_Rec2", Mix_Temp_Rec2 := "Mix_Temp_SP_Rec2", Mix_Temp_Tol_Rec2 := "Mix_Temp_Tol_Rec2", Mixing_Time_Rec2 := "Mix_Time_Rec2", Bottle_Size_Rec3 := "Bottle_Size_Rec3", Bottle_Number_Rec3 := "Bottle_Batch_Size_Rec3", Product_A_Rec3 := "ProdA_SP_Rec3", Product_A_Tol_Rec3 := "ProdA_Tol_Rec3", Product_B_Rec3 := "ProdB_SP_Rec3", Product_B_Tol_Rec3 := "ProdB_Tol_Rec3", Mix_Temp_Rec3 := "Mix_Temp_SP_Rec3", Mix_Temp_Tol_Rec3 := "Mix_Temp_Tol_Rec3", Mixing_Time_Rec3 := "Mix_Time_Rec3", "Recipe 1" := "Recipe_1", "Recipe 2" := "Recipe_2", Reset := "Reset_PB", "Recipe 3" := "Recipe_3", Bottle_Size =>, Bottle_Number =>, Product_A =>, Product_A_Tol =>, Product_B =>, Product_B_Tol =>, Mix_Temp =>, Mix_Temp_Tol =>, Mixing_Time =>, "Batch_Size_A+B" =>, Recipe_Selected_Out =>)
   END_RUNG
   // the same network as SCL:
   "Recipe Selection_DB"(Bottle_Size_Rec1 := "Bottle_Size_Rec1",   // "Recipe Selection"
                         Bottle_Number_Rec1 := "Bottle_Batch_Size_Rec1",
                         Product_A_Rec1 := "ProdA_SP_Rec1",
                         Product_A_Tol_Rec1 := "ProdA_Tol_Rec1",
                         Product_B_Rec1 := "ProdB_SP_Rec1",
                         Product_B_Tol_Rec1 := "ProdB_Tol_Rec1",
                         Mix_Temp_Rec1 := "Mix_Temp_SP_Rec1",
                         Mix_Temp_Tol_Rec1 := "Mix_Temp_Tol_Rec1",
                         Mixing_Time_Rec1 := "Mix_Time_Rec1",
                         Bottle_Size_Rec2 := "Bottle_Size_Rec2",
                         Bottle_Number_Rec2 := "Bottle_Batch_Size_Rec2",
                         Product_A_Rec2 := "ProdA_SP_Rec2",
                         Product_A_Tol_Rec2 := "ProdA_Tol_Rec2",
                         Product_B_Rec2 := "ProdB_SP_Rec2",
                         Product_B_Tol_Rec2 := "ProdB_Tol_Rec2",
                         Mix_Temp_Rec2 := "Mix_Temp_SP_Rec2",
                         Mix_Temp_Tol_Rec2 := "Mix_Temp_Tol_Rec2",
                         Mixing_Time_Rec2 := "Mix_Time_Rec2",
                         Bottle_Size_Rec3 := "Bottle_Size_Rec3",
                         Bottle_Number_Rec3 := "Bottle_Batch_Size_Rec3",
                         Product_A_Rec3 := "ProdA_SP_Rec3",
                         Product_A_Tol_Rec3 := "ProdA_Tol_Rec3",
                         Product_B_Rec3 := "ProdB_SP_Rec3",
                         Product_B_Tol_Rec3 := "ProdB_Tol_Rec3",
                         Mix_Temp_Rec3 := "Mix_Temp_SP_Rec3",
                         Mix_Temp_Tol_Rec3 := "Mix_Temp_Tol_Rec3",
                         Mixing_Time_Rec3 := "Mix_Time_Rec3",
                         "Recipe 1" := "Recipe_1",
                         "Recipe 2" := "Recipe_2",
                         Reset := "Reset_PB",
                         "Recipe 3" := "Recipe_3");
END_REGION

REGION Network 3: Process Sequence Diagram
   // Overview of the Automatic Mode process with conditions required for confirm the steps.
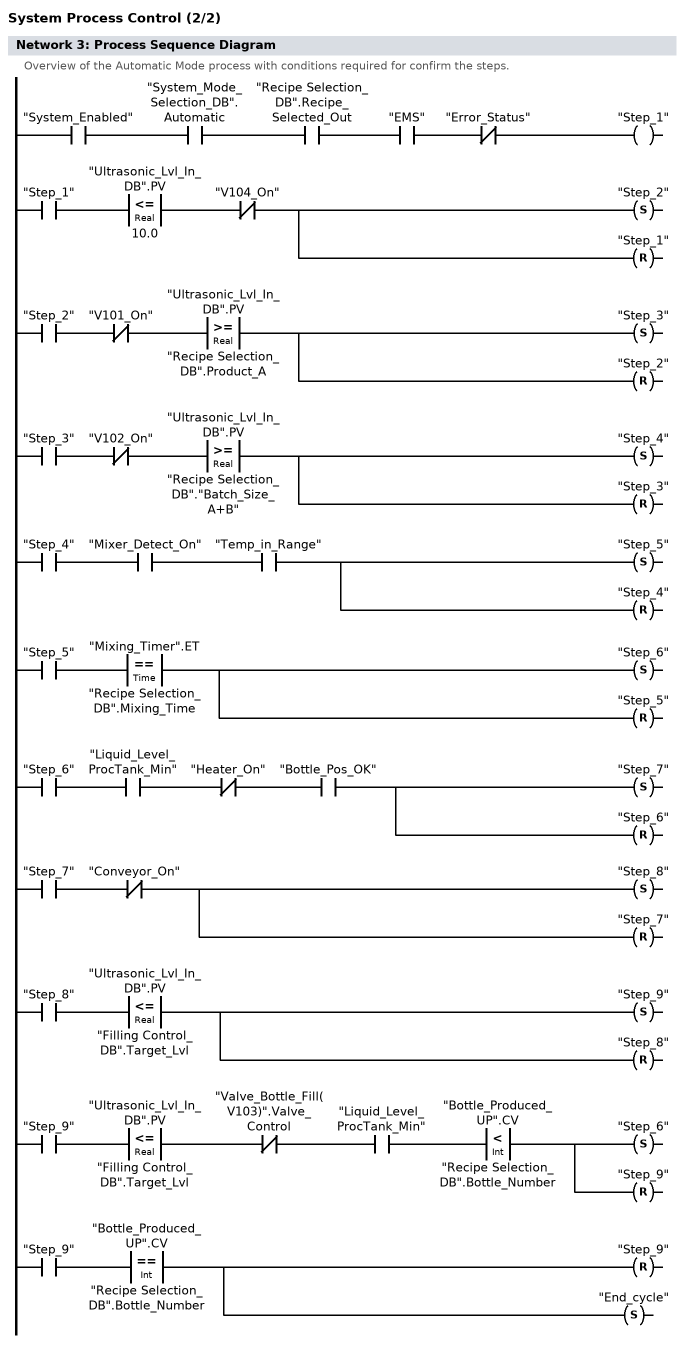
   RUNG wire#powerrail
      Contact( "System_Enabled" )
      Contact( "System_Mode_Selection_DB".Automatic )
      Contact( "Recipe Selection_DB".Recipe_Selected_Out )
      Contact( "EMS" )
      I_Contact( "Error_Status" )
      Coil( "Step_1" )
   END_RUNG
   RUNG wire#powerrail
      Contact( "Step_1" )
      { S7_Templates := "SrcType := Real" } LE_Contact(in1 := "Ultrasonic_Lvl_In_DB".PV, in2 := 10.0)
      I_Contact( "V104_On" )
      wire#w1
      S_Coil( "Step_2" )
   END_RUNG
   RUNG wire#w1
      R_Coil( "Step_1" )
   END_RUNG
   RUNG wire#powerrail
      Contact( "Step_2" )
      I_Contact( "V101_On" )
      { S7_Templates := "SrcType := Real" } GE_Contact(in1 := "Ultrasonic_Lvl_In_DB".PV, in2 := "Recipe Selection_DB".Product_A)
      wire#w2
      S_Coil( "Step_3" )
   END_RUNG
   RUNG wire#w2
      R_Coil( "Step_2" )
   END_RUNG
   RUNG wire#powerrail
      Contact( "Step_3" )
      I_Contact( "V102_On" )
      { S7_Templates := "SrcType := Real" } GE_Contact(in1 := "Ultrasonic_Lvl_In_DB".PV, in2 := "Recipe Selection_DB"."Batch_Size_A+B")
      wire#w3
      S_Coil( "Step_4" )
   END_RUNG
   RUNG wire#w3
      R_Coil( "Step_3" )
   END_RUNG
   RUNG wire#powerrail
      Contact( "Step_4" )
      Contact( "Mixer_Detect_On" )
      Contact( "Temp_in_Range" )
      wire#w4
      S_Coil( "Step_5" )
   END_RUNG
   RUNG wire#w4
      R_Coil( "Step_4" )
   END_RUNG
   RUNG wire#powerrail
      Contact( "Step_5" )
      { S7_Templates := "SrcType := Time" } EQ_Contact(in1 := "Mixing_Timer".ET, in2 := "Recipe Selection_DB".Mixing_Time)
      wire#w5
      S_Coil( "Step_6" )
   END_RUNG
   RUNG wire#w5
      R_Coil( "Step_5" )
   END_RUNG
   RUNG wire#powerrail
      Contact( "Step_6" )
      Contact( "Liquid_Level_ProcTank_Min" )
      I_Contact( "Heater_On" )
      Contact( "Bottle_Pos_OK" )
      wire#w6
      S_Coil( "Step_7" )
   END_RUNG
   RUNG wire#w6
      R_Coil( "Step_6" )
   END_RUNG
   RUNG wire#powerrail
      Contact( "Step_7" )
      I_Contact( "Conveyor_On" )
      wire#w7
      S_Coil( "Step_8" )
   END_RUNG
   RUNG wire#w7
      R_Coil( "Step_7" )
   END_RUNG
   RUNG wire#powerrail
      Contact( "Step_8" )
      { S7_Templates := "SrcType := Real" } LE_Contact(in1 := "Ultrasonic_Lvl_In_DB".PV, in2 := "Filling Control_DB".Target_Lvl)
      wire#w8
      S_Coil( "Step_9" )
   END_RUNG
   RUNG wire#w8
      R_Coil( "Step_8" )
   END_RUNG
   RUNG wire#powerrail
      Contact( "Step_9" )
      { S7_Templates := "SrcType := Real" } LE_Contact(in1 := "Ultrasonic_Lvl_In_DB".PV, in2 := "Filling Control_DB".Target_Lvl)
      I_Contact( "Valve_Bottle_Fill(V103)".Valve_Control )
      Contact( "Liquid_Level_ProcTank_Min" )
      { S7_Templates := "SrcType := Int" } LT_Contact(in1 := "Bottle_Produced_UP".CV, in2 := "Recipe Selection_DB".Bottle_Number)
      wire#w9
      S_Coil( "Step_6" )
   END_RUNG
   RUNG wire#w9
      R_Coil( "Step_9" )
   END_RUNG
   RUNG wire#powerrail
      Contact( "Step_9" )
      { S7_Templates := "SrcType := Int" } EQ_Contact(in1 := "Bottle_Produced_UP".CV, in2 := "Recipe Selection_DB".Bottle_Number)
      wire#w10
      R_Coil( "Step_9" )
   END_RUNG
   RUNG wire#w10
      S_Coil( "End_cycle" )
   END_RUNG
   // the same network as SCL:
   "Step_1" := "System_Enabled" AND "System_Mode_Selection_DB".Automatic AND "Recipe Selection_DB".Recipe_Selected_Out AND "EMS" AND NOT "Error_Status";
   IF "Step_1" AND ("Ultrasonic_Lvl_In_DB".PV <= 10.0) AND NOT "V104_On" THEN
       "Step_2" := TRUE;
       "Step_1" := FALSE;
   END_IF;
   IF "Step_2" AND NOT "V101_On" AND ("Ultrasonic_Lvl_In_DB".PV >= "Recipe Selection_DB".Product_A) THEN
       "Step_3" := TRUE;
       "Step_2" := FALSE;
   END_IF;
   IF "Step_3" AND NOT "V102_On" AND ("Ultrasonic_Lvl_In_DB".PV >= "Recipe Selection_DB"."Batch_Size_A+B") THEN
       "Step_4" := TRUE;
       "Step_3" := FALSE;
   END_IF;
   IF "Step_4" AND "Mixer_Detect_On" AND "Temp_in_Range" THEN
       "Step_5" := TRUE;
       "Step_4" := FALSE;
   END_IF;
   IF "Step_5" AND ("Mixing_Timer".ET = "Recipe Selection_DB".Mixing_Time) THEN
       "Step_6" := TRUE;
       "Step_5" := FALSE;
   END_IF;
   IF "Step_6" AND "Liquid_Level_ProcTank_Min" AND NOT "Heater_On" AND "Bottle_Pos_OK" THEN
       "Step_7" := TRUE;
       "Step_6" := FALSE;
   END_IF;
   IF "Step_7" AND NOT "Conveyor_On" THEN
       "Step_8" := TRUE;
       "Step_7" := FALSE;
   END_IF;
   IF "Step_8" AND ("Ultrasonic_Lvl_In_DB".PV <= "Filling Control_DB".Target_Lvl) THEN
       "Step_9" := TRUE;
       "Step_8" := FALSE;
   END_IF;
   IF "Step_9" AND ("Ultrasonic_Lvl_In_DB".PV <= "Filling Control_DB".Target_Lvl) AND NOT "Valve_Bottle_Fill(V103)".Valve_Control AND "Liquid_Level_ProcTank_Min" AND ("Bottle_Produced_UP".CV < "Recipe Selection_DB".Bottle_Number) THEN
       "Step_6" := TRUE;
       "Step_9" := FALSE;
   END_IF;
   #_w1 := "Step_9" AND ("Bottle_Produced_UP".CV = "Recipe Selection_DB".Bottle_Number);
   IF #_w1 THEN
       "Step_9" := FALSE;
       "End_cycle" := TRUE;
   END_IF;
END_REGION
END_FUNCTION

FUNCTION "Mixing Tank Processes" : Void   // FC2, LAD
{ S7_Optimized_Access := 'TRUE' }
VERSION : 0.1
// This function manages the processes relating to the Mixing Tank:
// - Filling in Mixing Tank with Product A and B.
// - Liquid Management in the Mixing Tank.
// - Purging Mixing Tank.
   VAR_TEMP   // added for the SCL form of the ladder/FBD networks
      _w1 : Bool;
   END_VAR
BEGIN

REGION Network 1: Ultrasonic Analogue Sensor.
   // Reading and Scaling Analogue values from the Ultrasonic level Sensor.
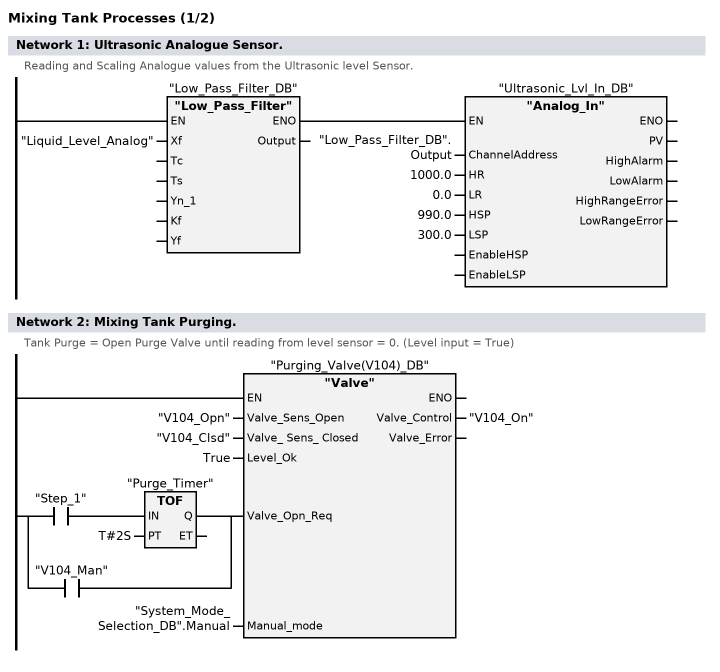
   RUNG wire#powerrail
      "Low_Pass_Filter_DB"(Xf := "Liquid_Level_Analog", Tc :=, Ts :=, Yn_1 :=, Kf :=, Yf :=, Output =>)
      "Ultrasonic_Lvl_In_DB"(ChannelAddress := "Low_Pass_Filter_DB".Output, HR := 1000.0, LR := 0.0, HSP := 990.0, LSP := 300.0, EnableHSP :=, EnableLSP :=, PV =>, HighAlarm =>, LowAlarm =>, HighRangeError =>, LowRangeError =>)
   END_RUNG
   // the same network as SCL:
   "Low_Pass_Filter_DB"(Xf := "Liquid_Level_Analog", ENO => #_w1);   // "Low_Pass_Filter"
   IF #_w1 THEN
       "Ultrasonic_Lvl_In_DB"(ChannelAddress := "Low_Pass_Filter_DB".Output,   // "Analog_In"
                              HR := 1000.0,
                              LR := 0.0,
                              HSP := 990.0,
                              LSP := 300.0);
   END_IF;
END_REGION

REGION Network 2: Mixing Tank Purging.
   // Tank Purge = Open Purge Valve until reading from level sensor = 0. (Level input = True)
   "Purge_Timer".TOF(IN := "Step_1", PT := T#2S);
   "Purging_Valve(V104)_DB"(Valve_Sens_Open := "V104_Opn",   // "Valve"
                           "Valve_ Sens_ Closed" := "V104_Clsd",
                           Level_Ok := True,
                           Valve_Opn_Req := "Purge_Timer".Q OR "V104_Man",
                           Manual_mode := "System_Mode_Selection_DB".Manual,
                           Valve_Control => "V104_On");
END_REGION

REGION Network 3: Preparing Product Mix.
   // Adding Product A then Product B; Once desired Level reached and Minimum Level Ok = Products Ready. // UPDATE TO TAKE TOLERANCE INTO ACCOUNT (IN_RANGE).
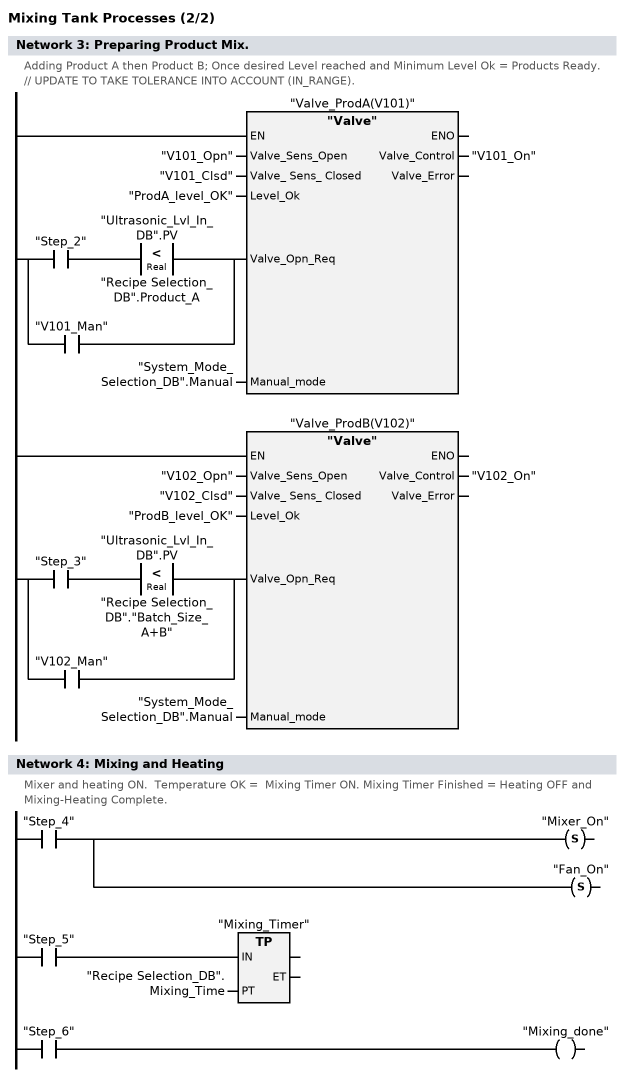
   RUNG wire#powerrail
      "Valve_ProdA(V101)"(Valve_Opn_Req := wire#w1, Valve_Sens_Open := "V101_Opn", "Valve_ Sens_ Closed" := "V101_Clsd", Level_Ok := "ProdA_level_OK", Manual_mode := "System_Mode_Selection_DB".Manual, Valve_Control => "V101_On", Valve_Error =>)
   END_RUNG
   RUNG wire#powerrail
      Contact( "Step_2" )
      { S7_Templates := "SrcType := Real" } LT_Contact(in1 := "Ultrasonic_Lvl_In_DB".PV, in2 := "Recipe Selection_DB".Product_A)
   END_RUNG wire#w1
   RUNG wire#powerrail
      Contact( "V101_Man" )
   END_RUNG wire#w1
   RUNG wire#powerrail
      "Valve_ProdB(V102)"(Valve_Opn_Req := wire#w2, Valve_Sens_Open := "V102_Opn", "Valve_ Sens_ Closed" := "V102_Clsd", Level_Ok := "ProdB_level_OK", Manual_mode := "System_Mode_Selection_DB".Manual, Valve_Control => "V102_On", Valve_Error =>)
   END_RUNG
   RUNG wire#powerrail
      Contact( "Step_3" )
      { S7_Templates := "SrcType := Real" } LT_Contact(in1 := "Ultrasonic_Lvl_In_DB".PV, in2 := "Recipe Selection_DB"."Batch_Size_A+B")
   END_RUNG wire#w2
   RUNG wire#powerrail
      Contact( "V102_Man" )
   END_RUNG wire#w2
   // the same network as SCL:
   "Valve_ProdA(V101)"(Valve_Sens_Open := "V101_Opn",   // "Valve"
                       "Valve_ Sens_ Closed" := "V101_Clsd",
                       Level_Ok := "ProdA_level_OK",
                       Valve_Opn_Req := ("Step_2" AND ("Ultrasonic_Lvl_In_DB".PV < "Recipe Selection_DB".Product_A)) OR "V101_Man",
                       Manual_mode := "System_Mode_Selection_DB".Manual,
                       Valve_Control => "V101_On");
   "Valve_ProdB(V102)"(Valve_Sens_Open := "V102_Opn",   // "Valve"
                       "Valve_ Sens_ Closed" := "V102_Clsd",
                       Level_Ok := "ProdB_level_OK",
                       Valve_Opn_Req := ("Step_3" AND ("Ultrasonic_Lvl_In_DB".PV < "Recipe Selection_DB"."Batch_Size_A+B")) OR "V102_Man",
                       Manual_mode := "System_Mode_Selection_DB".Manual,
                       Valve_Control => "V102_On");
END_REGION

REGION Network 4: Mixing and Heating
   // Mixer and heating ON.  Temperature OK =  Mixing Timer ON. Mixing Timer Finished = Heating OFF and Mixing-Heating Complete.
   IF "Step_4" THEN
       "Mixer_On" := TRUE;
       "Fan_On" := TRUE;
   END_IF;
   "Mixing_Timer".TP(IN := "Step_5", PT := "Recipe Selection_DB".Mixing_Time);
   "Mixing_done" := "Step_6";
END_REGION
END_FUNCTION

FUNCTION "Bottle Filling Conveyor Process" : Void   // FC3, LAD
TITLE = Conveyor and Bottle Filling Processes
{ S7_Optimized_Access := 'TRUE' }
VERSION : 0.1
// This Function manages the conveyor and bottle filling process:
// - Conveyor Control.
// - Bottle filling.
BEGIN

REGION Network 1: Conveyor Control
   // Conveyor Control: The conveyor is activated by the end of the mixing cycle or by the end of a bottle filling. The speed of the conveyor is set by by the analogue output. The conveyor is stopped by the bottle being in position.
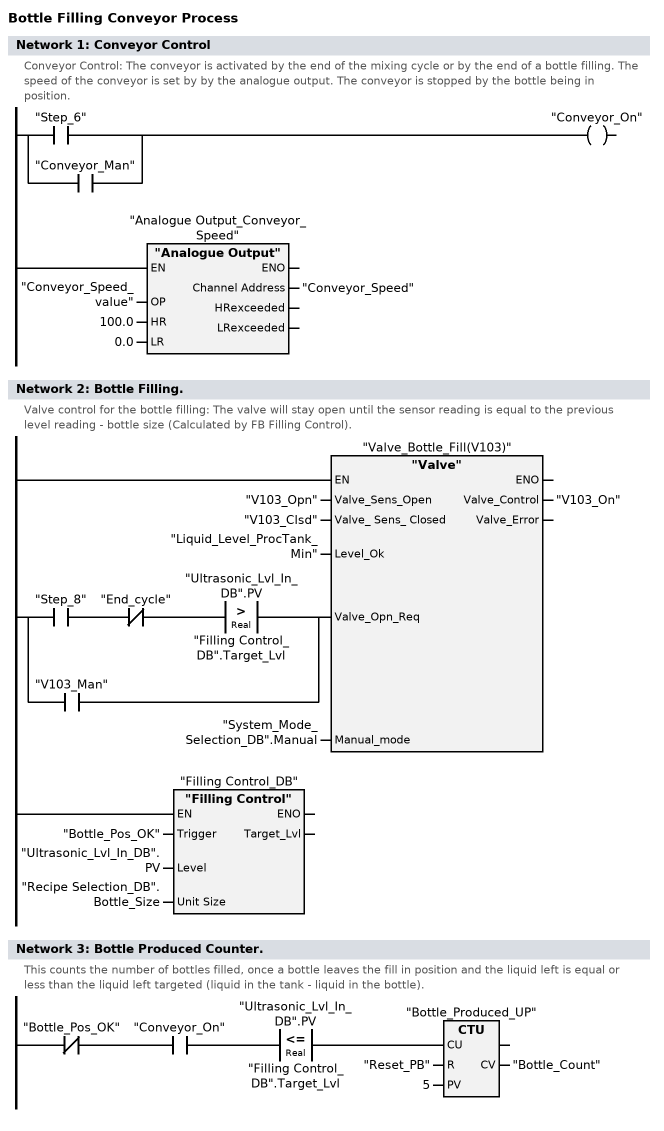
   RUNG wire#powerrail
      Contact( "Step_6" )
      wire#w1
      Coil( "Conveyor_On" )
   END_RUNG
   RUNG wire#powerrail
      Contact( "Conveyor_Man" )
   END_RUNG wire#w1
   RUNG wire#powerrail
      "Analogue Output_Conveyor_Speed"(OP := "Conveyor_Speed_value", HR := 100.0, LR := 0.0, "Channel Address" => "Conveyor_Speed", HRexceeded =>, LRexceeded =>)
   END_RUNG
   // the same network as SCL:
   "Conveyor_On" := "Step_6" OR "Conveyor_Man";
   "Analogue Output_Conveyor_Speed"(OP := "Conveyor_Speed_value",   // "Analogue Output"
                           HR := 100.0,
                           LR := 0.0,
                           "Channel Address" => "Conveyor_Speed");
END_REGION

REGION Network 2: Bottle Filling.
   // Valve control for the bottle filling: The valve will stay open until the sensor reading is equal to the previous level reading - bottle size (Calculated by FB Filling Control).
   RUNG wire#powerrail
      "Valve_Bottle_Fill(V103)"(Valve_Opn_Req := wire#w1, Valve_Sens_Open := "V103_Opn", "Valve_ Sens_ Closed" := "V103_Clsd", Level_Ok := "Liquid_Level_ProcTank_Min", Manual_mode := "System_Mode_Selection_DB".Manual, Valve_Control => "V103_On", Valve_Error =>)
   END_RUNG
   RUNG wire#powerrail
      Contact( "Step_8" )
      I_Contact( "End_cycle" )
      { S7_Templates := "SrcType := Real" } GT_Contact(in1 := "Ultrasonic_Lvl_In_DB".PV, in2 := "Filling Control_DB".Target_Lvl)
   END_RUNG wire#w1
   RUNG wire#powerrail
      Contact( "V103_Man" )
   END_RUNG wire#w1
   RUNG wire#powerrail
      "Filling Control_DB"(Trigger := "Bottle_Pos_OK", Level := "Ultrasonic_Lvl_In_DB".PV, "Unit Size" := "Recipe Selection_DB".Bottle_Size, Target_Lvl =>)
   END_RUNG
   // the same network as SCL:
   "Valve_Bottle_Fill(V103)"(Valve_Sens_Open := "V103_Opn",   // "Valve"
                           "Valve_ Sens_ Closed" := "V103_Clsd",
                           Level_Ok := "Liquid_Level_ProcTank_Min",
                           Valve_Opn_Req := ("Step_8" AND NOT "End_cycle" AND ("Ultrasonic_Lvl_In_DB".PV > "Filling Control_DB".Target_Lvl)) OR "V103_Man",
                           Manual_mode := "System_Mode_Selection_DB".Manual,
                           Valve_Control => "V103_On");
   "Filling Control_DB"(Trigger := "Bottle_Pos_OK",   // "Filling Control"
                        Level := "Ultrasonic_Lvl_In_DB".PV,
                        "Unit Size" := "Recipe Selection_DB".Bottle_Size);
END_REGION

REGION Network 3: Bottle Produced Counter.
   // This counts the number of bottles filled, once a bottle leaves the fill in position and the liquid left is equal or less than the liquid left targeted (liquid in the tank - liquid in the bottle).
   "Bottle_Produced_UP".CTU(CU := NOT "Bottle_Pos_OK" AND "Conveyor_On" AND ("Ultrasonic_Lvl_In_DB".PV <= "Filling Control_DB".Target_Lvl),
                           R := "Reset_PB",
                           PV := 5,
                           CV => "Bottle_Count");
END_REGION
END_FUNCTION

FUNCTION "Error Management" : Void   // FC4, LAD
TITLE = Error Management and Machine Reset.
{ S7_Optimized_Access := 'TRUE' }
VERSION : 0.1
// This Block Manages the error cases and Reset function:
// - If Stop, EMS or Reset are hit the machine will stop and reset.
// - If the heating element is on and the liquid level is below 300L or the level switch is off an error will be triggered.
// - Product A and B liquid Level Error.
// - At the bottling stage if the conveyor is on for a minute with no bottles the machine will stop.
// - If the level for each product A and B goes above or below the levels of tolerances an error will be triggered.
   VAR_TEMP   // added for the SCL form of the ladder/FBD networks
      _w1 : Bool;
   END_VAR
BEGIN

REGION Network 1: Error Management Valves
   // If any of the valve control functions return an error the error_status is set.
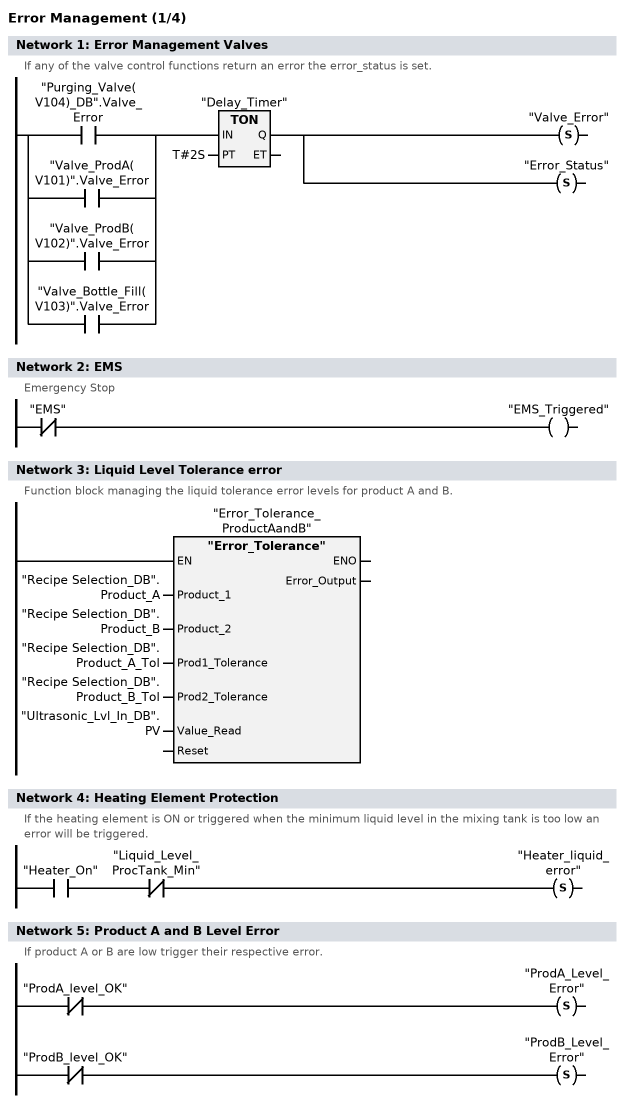
   "Delay_Timer".TON(IN := "Purging_Valve(V104)_DB".Valve_Error OR "Valve_ProdA(V101)".Valve_Error OR "Valve_ProdB(V102)".Valve_Error OR "Valve_Bottle_Fill(V103)".Valve_Error,
                     PT := T#2S);
   IF "Delay_Timer".Q THEN
       "Valve_Error" := TRUE;
       "Error_Status" := TRUE;
   END_IF;
END_REGION

REGION Network 2: EMS
   // Emergency Stop
   RUNG wire#powerrail
      I_Contact( "EMS" )
      Coil( "EMS_Triggered" )
   END_RUNG
   // the same network as SCL:
   "EMS_Triggered" := NOT "EMS";
END_REGION

REGION Network 3: Liquid Level Tolerance error
   // Function block managing the liquid tolerance error levels for product A and B.
   RUNG wire#powerrail
      "Error_Tolerance_ProductAandB"(Product_1 := "Recipe Selection_DB".Product_A, Product_2 := "Recipe Selection_DB".Product_B, Prod1_Tolerance := "Recipe Selection_DB".Product_A_Tol, Prod2_Tolerance := "Recipe Selection_DB".Product_B_Tol, Value_Read := "Ultrasonic_Lvl_In_DB".PV, Reset :=, Error_Output =>)
   END_RUNG
   // the same network as SCL:
   "Error_Tolerance_ProductAandB"(Product_1 := "Recipe Selection_DB".Product_A,   // "Error_Tolerance"
                           Product_2 := "Recipe Selection_DB".Product_B,
                           Prod1_Tolerance := "Recipe Selection_DB".Product_A_Tol,
                           Prod2_Tolerance := "Recipe Selection_DB".Product_B_Tol,
                           Value_Read := "Ultrasonic_Lvl_In_DB".PV);
END_REGION

REGION Network 4: Heating Element Protection
   // If the heating element is ON or triggered when the minimum liquid level in the mixing tank is too low an error will be triggered.
   RUNG wire#powerrail
      Contact( "Heater_On" )
      I_Contact( "Liquid_Level_ProcTank_Min" )
      S_Coil( "Heater_liquid_error" )
   END_RUNG
   // the same network as SCL:
   IF "Heater_On" AND NOT "Liquid_Level_ProcTank_Min" THEN "Heater_liquid_error" := TRUE; END_IF;
END_REGION

REGION Network 5: Product A and B Level Error
   // If product A or B are low trigger their respective error.
   RUNG wire#powerrail
      I_Contact( "ProdA_level_OK" )
      S_Coil( "ProdA_Level_Error" )
   END_RUNG
   RUNG wire#powerrail
      I_Contact( "ProdB_level_OK" )
      S_Coil( "ProdB_Level_Error" )
   END_RUNG
   // the same network as SCL:
   IF NOT "ProdA_level_OK" THEN "ProdA_Level_Error" := TRUE; END_IF;
   IF NOT "ProdB_level_OK" THEN "ProdB_Level_Error" := TRUE; END_IF;
END_REGION

REGION Network 6: Tank Overflow Error.
   // If the supply valves are on and  the sensor reading goes over 998 Litres the error will trigger
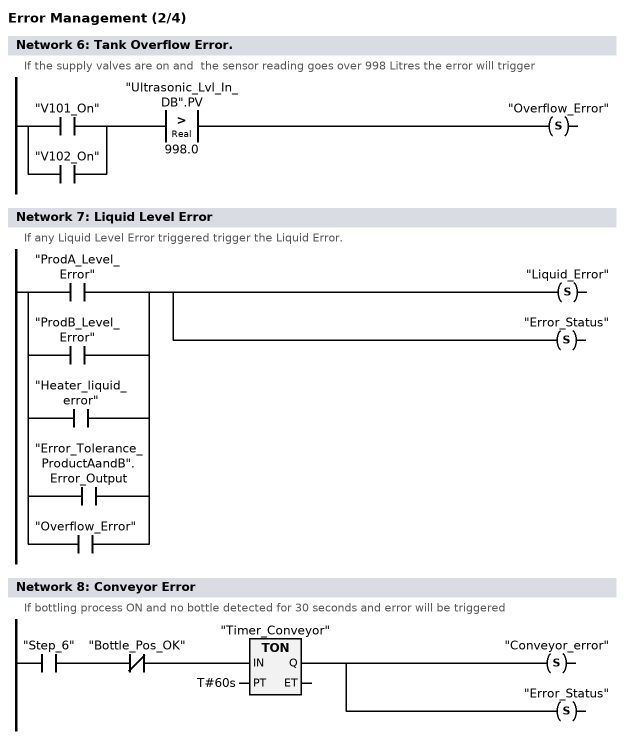
   RUNG wire#powerrail
      Contact( "V101_On" )
      wire#w1
      { S7_Templates := "SrcType := Real" } GT_Contact(in1 := "Ultrasonic_Lvl_In_DB".PV, in2 := 998.0)
      S_Coil( "Overflow_Error" )
   END_RUNG
   RUNG wire#powerrail
      Contact( "V102_On" )
   END_RUNG wire#w1
   // the same network as SCL:
   IF ("V101_On" OR "V102_On") AND ("Ultrasonic_Lvl_In_DB".PV > 998.0) THEN "Overflow_Error" := TRUE; END_IF;
END_REGION

REGION Network 7: Liquid Level Error
   // If any Liquid Level Error triggered trigger the Liquid Error.
   RUNG wire#powerrail
      Contact( "ProdA_Level_Error" )
      wire#w1
      S_Coil( "Liquid_Error" )
   END_RUNG
   RUNG wire#powerrail
      Contact( "ProdB_Level_Error" )
   END_RUNG wire#w1
   RUNG wire#powerrail
      Contact( "Heater_liquid_error" )
   END_RUNG wire#w1
   RUNG wire#powerrail
      Contact( "Error_Tolerance_ProductAandB".Error_Output )
   END_RUNG wire#w1
   RUNG wire#powerrail
      Contact( "Overflow_Error" )
   END_RUNG wire#w1
   RUNG wire#w1
      S_Coil( "Error_Status" )
   END_RUNG
   // the same network as SCL:
   IF "ProdA_Level_Error" OR "ProdB_Level_Error" OR "Heater_liquid_error" OR "Error_Tolerance_ProductAandB".Error_Output OR "Overflow_Error" THEN
       "Liquid_Error" := TRUE;
       "Error_Status" := TRUE;
   END_IF;
END_REGION

REGION Network 8: Conveyor Error
   // If bottling process ON and no bottle detected for 30 seconds and error will be triggered
   "Timer_Conveyor".TON(IN := "Step_6" AND NOT "Bottle_Pos_OK", PT := T#60s);
   IF "Timer_Conveyor".Q THEN
       "Conveyor_error" := TRUE;
       "Error_Status" := TRUE;
   END_IF;
END_REGION

REGION Network 9: System Reset
   // System can be reset by: Reset_PB, EMS and Stop_PB.
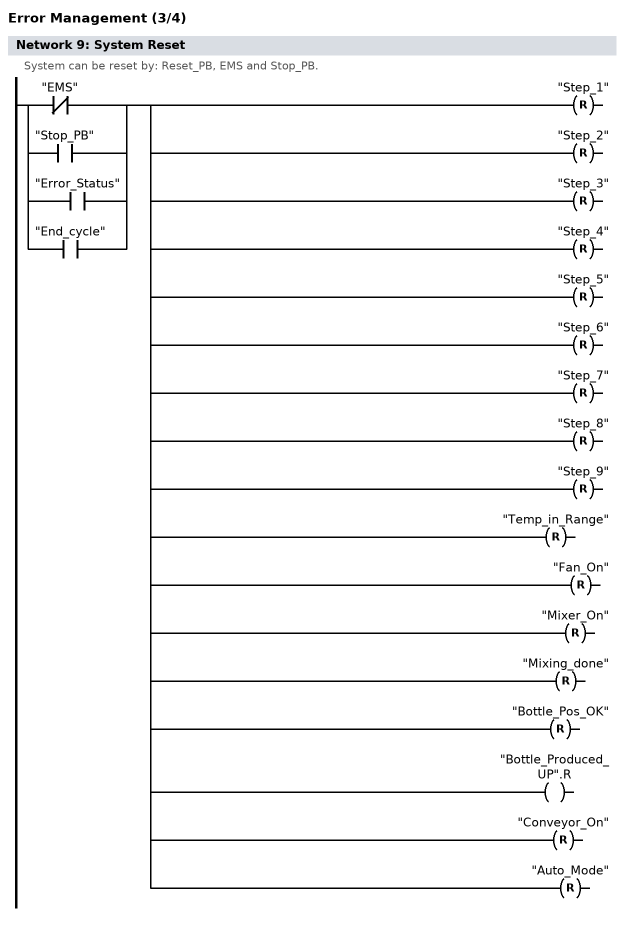
   RUNG wire#powerrail
      I_Contact( "EMS" )
      wire#w1
      R_Coil( "Step_1" )
   END_RUNG
   RUNG wire#powerrail
      Contact( "Stop_PB" )
   END_RUNG wire#w1
   RUNG wire#powerrail
      Contact( "Error_Status" )
   END_RUNG wire#w1
   RUNG wire#powerrail
      Contact( "End_cycle" )
   END_RUNG wire#w1
   RUNG wire#w1
      R_Coil( "Step_2" )
   END_RUNG
   RUNG wire#w1
      R_Coil( "Step_3" )
   END_RUNG
   RUNG wire#w1
      R_Coil( "Step_4" )
   END_RUNG
   RUNG wire#w1
      R_Coil( "Step_5" )
   END_RUNG
   RUNG wire#w1
      R_Coil( "Step_6" )
   END_RUNG
   RUNG wire#w1
      R_Coil( "Step_7" )
   END_RUNG
   RUNG wire#w1
      R_Coil( "Step_8" )
   END_RUNG
   RUNG wire#w1
      R_Coil( "Step_9" )
   END_RUNG
   RUNG wire#w1
      R_Coil( "Temp_in_Range" )
   END_RUNG
   RUNG wire#w1
      R_Coil( "Fan_On" )
   END_RUNG
   RUNG wire#w1
      R_Coil( "Mixer_On" )
   END_RUNG
   RUNG wire#w1
      R_Coil( "Mixing_done" )
   END_RUNG
   RUNG wire#w1
      R_Coil( "Bottle_Pos_OK" )
   END_RUNG
   RUNG wire#w1
      Coil( "Bottle_Produced_UP".R )
   END_RUNG
   RUNG wire#w1
      R_Coil( "Conveyor_On" )
   END_RUNG
   RUNG wire#w1
      R_Coil( "Auto_Mode" )
   END_RUNG
   // the same network as SCL:
   #_w1 := NOT "EMS" OR "Stop_PB" OR "Error_Status" OR "End_cycle";
   IF #_w1 THEN
       "Step_1" := FALSE;
       "Step_2" := FALSE;
       "Step_3" := FALSE;
       "Step_4" := FALSE;
       "Step_5" := FALSE;
       "Step_6" := FALSE;
       "Step_7" := FALSE;
       "Step_8" := FALSE;
       "Step_9" := FALSE;
       "Temp_in_Range" := FALSE;
       "Fan_On" := FALSE;
       "Mixer_On" := FALSE;
       "Mixing_done" := FALSE;
       "Bottle_Pos_OK" := FALSE;
   END_IF;
   "Bottle_Produced_UP".R := #_w1;
   IF #_w1 THEN
       "Conveyor_On" := FALSE;
       "Auto_Mode" := FALSE;
   END_IF;
END_REGION

REGION Network 10: Error Reset
   // Error Status can be reset using the Reset button.
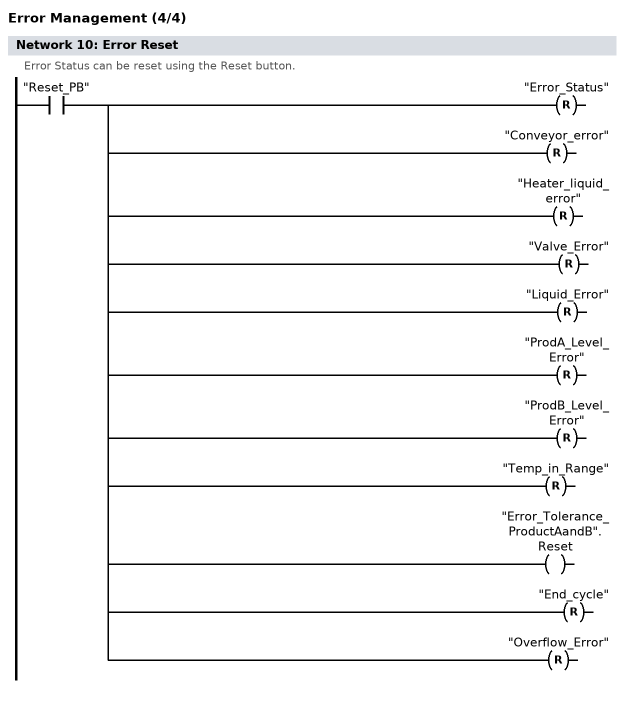
   RUNG wire#powerrail
      Contact( "Reset_PB" )
      wire#w1
      R_Coil( "Error_Status" )
   END_RUNG
   RUNG wire#w1
      R_Coil( "Conveyor_error" )
   END_RUNG
   RUNG wire#w1
      R_Coil( "Heater_liquid_error" )
   END_RUNG
   RUNG wire#w1
      R_Coil( "Valve_Error" )
   END_RUNG
   RUNG wire#w1
      R_Coil( "Liquid_Error" )
   END_RUNG
   RUNG wire#w1
      R_Coil( "ProdA_Level_Error" )
   END_RUNG
   RUNG wire#w1
      R_Coil( "ProdB_Level_Error" )
   END_RUNG
   RUNG wire#w1
      R_Coil( "Temp_in_Range" )
   END_RUNG
   RUNG wire#w1
      Coil( "Error_Tolerance_ProductAandB".Reset )
   END_RUNG
   RUNG wire#w1
      R_Coil( "End_cycle" )
   END_RUNG
   RUNG wire#w1
      R_Coil( "Overflow_Error" )
   END_RUNG
   // the same network as SCL:
   IF "Reset_PB" THEN
       "Error_Status" := FALSE;
       "Conveyor_error" := FALSE;
       "Heater_liquid_error" := FALSE;
       "Valve_Error" := FALSE;
       "Liquid_Error" := FALSE;
       "ProdA_Level_Error" := FALSE;
       "ProdB_Level_Error" := FALSE;
       "Temp_in_Range" := FALSE;
   END_IF;
   "Error_Tolerance_ProductAandB".Reset := "Reset_PB";
   IF "Reset_PB" THEN
       "End_cycle" := FALSE;
       "Overflow_Error" := FALSE;
   END_IF;
END_REGION
END_FUNCTION

FUNCTION "Temperature Management" : Void   // FC5, LAD
{ S7_Optimized_Access := 'TRUE' }
VERSION : 0.1
// This function manages the Temperature Functionalities of the programme:
// - Reading and Scaling an Analogue Value.
// - Temperature in range check.
   VAR_TEMP
      Temp_Limit_Low_Range : Real;
      Temp_Limit_High_Range : Real;
   END_VAR
BEGIN

REGION Network 1: Analogue Temperature Input
   // The Function Block reads and Scales the analogue values between -200 and 200°C. Also Provides alarms when reading exceed 150°C or goes below -100°C.
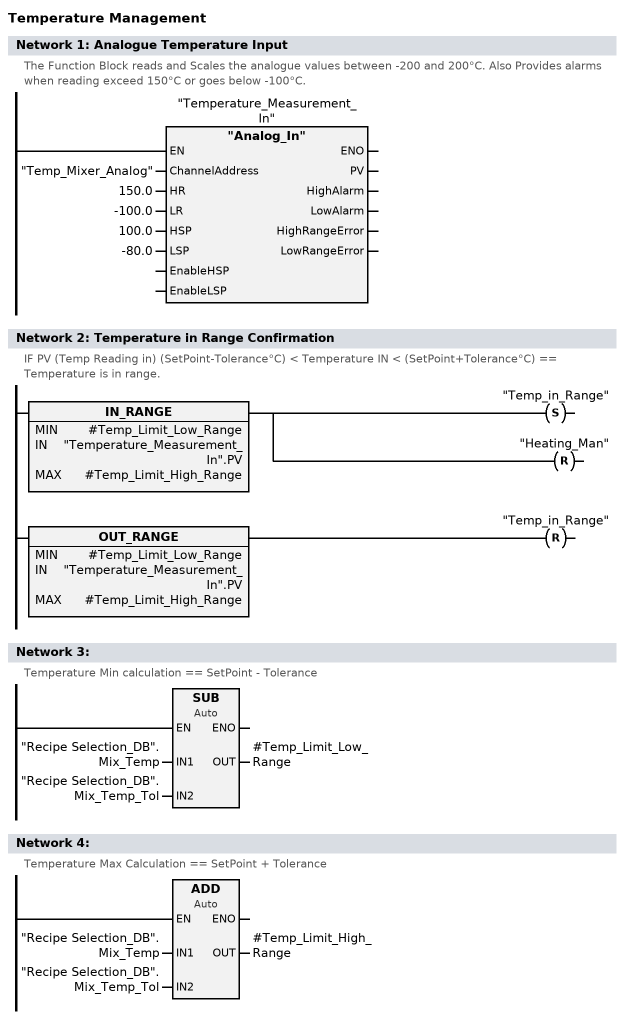
   RUNG wire#powerrail
      "Temperature_Measurement_In"(ChannelAddress := "Temp_Mixer_Analog", HR := 150.0, LR := -100.0, HSP := 100.0, LSP := -80.0, EnableHSP :=, EnableLSP :=, PV =>, HighAlarm =>, LowAlarm =>, HighRangeError =>, LowRangeError =>)
   END_RUNG
   // the same network as SCL:
   "Temperature_Measurement_In"(ChannelAddress := "Temp_Mixer_Analog",   // "Analog_In"
                           HR := 150.0,
                           LR := -100.0,
                           HSP := 100.0,
                           LSP := -80.0);
END_REGION

REGION Network 2: Temperature in Range Confirmation
   // IF PV (Temp Reading in) (SetPoint-Tolerance°C) < Temperature IN < (SetPoint+Tolerance°C) == Temperature is in range.
   IF (#Temp_Limit_Low_Range <= "Temperature_Measurement_In".PV) AND ("Temperature_Measurement_In".PV <= #Temp_Limit_High_Range) THEN
       "Temp_in_Range" := TRUE;
       "Heating_Man" := FALSE;
   END_IF;
   IF ("Temperature_Measurement_In".PV < #Temp_Limit_Low_Range) OR ("Temperature_Measurement_In".PV > #Temp_Limit_High_Range) THEN
       "Temp_in_Range" := FALSE;
   END_IF;
END_REGION

REGION Network 3
   // Temperature Min calculation == SetPoint - Tolerance
   RUNG wire#powerrail
      { S7_GenerateENO := "TRUE" } Sub(in1 := "Recipe Selection_DB".Mix_Temp, in2 := "Recipe Selection_DB".Mix_Temp_Tol, out => #Temp_Limit_Low_Range)
   END_RUNG
   // the same network as SCL:
   #Temp_Limit_Low_Range := "Recipe Selection_DB".Mix_Temp - "Recipe Selection_DB".Mix_Temp_Tol;
END_REGION

REGION Network 4
   // Temperature Max Calculation == SetPoint + Tolerance
   RUNG wire#powerrail
      { S7_GenerateENO := "TRUE" } Add(in1 := "Recipe Selection_DB".Mix_Temp, in2 := "Recipe Selection_DB".Mix_Temp_Tol, out => #Temp_Limit_High_Range)
   END_RUNG
   // the same network as SCL:
   #Temp_Limit_High_Range := "Recipe Selection_DB".Mix_Temp + "Recipe Selection_DB".Mix_Temp_Tol;
END_REGION
END_FUNCTION

ORGANIZATION_BLOCK "Main"   // OB1, LAD, ProgramCycle
TITLE = "Main Program Sweep (Cycle)"
{ S7_Optimized_Access := 'TRUE' }
VERSION : 0.1
   VAR_TEMP   // added for the SCL form of the ladder/FBD networks
      _w1 : Bool;
   END_VAR
BEGIN

REGION Network 1
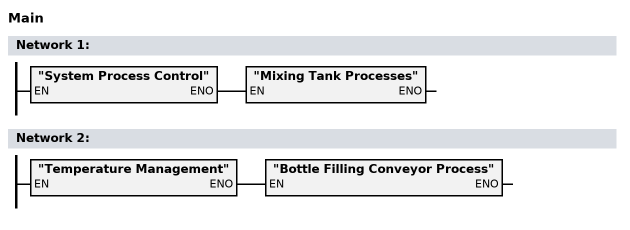
   RUNG wire#powerrail
      "System Process Control"()
      "Mixing Tank Processes"()
   END_RUNG
   // the same network as SCL:
   "System Process Control"(ENO => #_w1);
   IF #_w1 THEN "Mixing Tank Processes"(); END_IF;
END_REGION

REGION Network 2
   RUNG wire#powerrail
      "Temperature Management"()
      "Bottle Filling Conveyor Process"()
   END_RUNG
   // the same network as SCL:
   "Temperature Management"(ENO => #_w1);
   IF #_w1 THEN "Bottle Filling Conveyor Process"(); END_IF;
END_REGION
END_ORGANIZATION_BLOCK

ORGANIZATION_BLOCK "Cyclic interrupt"   // OB30, LAD, CyclicInterrupt
{ S7_Optimized_Access := 'TRUE' }
VERSION : 0.1
BEGIN

REGION Network 1: Temperature Control
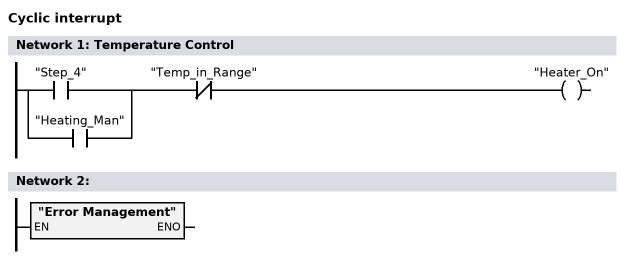
   RUNG wire#powerrail
      Contact( "Step_4" )
      wire#w1
      I_Contact( "Temp_in_Range" )
      Coil( "Heater_On" )
   END_RUNG
   RUNG wire#powerrail
      Contact( "Heating_Man" )
   END_RUNG wire#w1
   // the same network as SCL:
   "Heater_On" := ("Step_4" OR "Heating_Man") AND NOT "Temp_in_Range";
END_REGION

REGION Network 2
   RUNG wire#powerrail
      "Error Management"()
   END_RUNG
   // the same network as SCL:
   "Error Management"();
END_REGION
END_ORGANIZATION_BLOCK

(* ===== HMI "HMI_RT_1" =====
system functions are stored by id; their names below are inferred from use
connection "HMI_Connection_1": ETHERNET, SMART_S7_1200_OMS
connection "HMI_Connection_2": ETHERNET, SMART_S7_1200_OMS

HMI tags "Default tag table"
   "TankSimulator_DB_Level" : Real = PLC TankSimulator_DB.Level, 1 s
   "V101_LimitOpenLSW" : Bool = PLC V101.LimitOpenLSW, 1 s
   "V101_LimitCloseLSW" : Bool = PLC V101.LimitCloseLSW, 1 s
   "V102_LimitOpenLSW" : Bool = PLC V102.LimitOpenLSW, 1 s
   "V102_LimitCloseLSW" : Bool = PLC V102.LimitCloseLSW, 1 s
   "V104_LimitOpenLSW" : Bool = PLC V104.LimitOpenLSW, 1 s
   "V104_LimitCloseLSW" : Bool = PLC V104.LimitCloseLSW, 1 s
   "V103_LimitOpenLSW" : Bool = PLC V103.LimitOpenLSW, 1 s
   "V103_LimitCloseLSW" : Bool = PLC V103.LimitCloseLSW, 1 s
   "MixerRunning" : Bool = PLC MixerRunning AT %Q1.4, 1 s
   "HeatLevel" : Bool = PLC MinimumHeatTankLevel AT %Q1.0, 1 s
   "V101_FaultEnable" : Bool = PLC V101.FaultEnable, 1 s
   "V102_FaultEnable" : Bool = PLC V102.FaultEnable, 1 s
   "V103_FaultEnable" : Bool = PLC V103.FaultEnable, 1 s
   "V104_FaultEnable" : Bool = PLC V104.FaultEnable, 1 s
   "V104_OpTime" : Int = PLC V104.OpTime, 1 s
   "Start_PB" : Bool = PLC Start_PB AT %M10.0, 1 s
   "Stop_PB" : Bool = PLC Stop_PB AT %M11.0, 1 s
   "Reset_PB" : Bool = PLC Reset_PB AT %M15.0, 1 s
   "Auto_Mode" : Bool = PLC Auto_Mode AT %M12.0, 1 s
   "Manual_Mode" : Bool = PLC Manual_Mode AT %M13.0, 1 s
   "Recipe_1" : Bool = PLC Recipe_1 AT %M118.0, 1 s
   "Recipe_2" : Bool = PLC Recipe_2 AT %M119.0, 1 s
   "Recipe_3" : Bool = PLC Recipe_3 AT %M120.0, 1 s
   "Bottle_Size_Rec1" : Int = PLC Bottle_Size_Rec1 AT %MW114, 1 s
   "Bottle_Size_Rec2" : Int = PLC Bottle_Size_Rec2 AT %MW134, 1 s
   "Bottle_Size_Rec3" : Int = PLC Bottle_Size_Rec3 AT %MW152, 1 s
   "Bottle_Batch_Size_Rec1" : Int = PLC Bottle_Batch_Size_Rec1 AT %MW116, 1 s
   "Bottle_Batch_Size_Rec2" : Int = PLC Bottle_Batch_Size_Rec2 AT %MW136, 1 s
   "Bottle_Batch_Size_Rec3" : Int = PLC Bottle_Batch_Size_Rec3 AT %MW154, 1 s
   "ProdA_SP_Rec1" : Int = PLC ProdA_SP_Rec1 AT %MW100, 1 s
   "ProdA_Tol_Rec1" : Int = PLC ProdA_Tol_Rec1 AT %MW104, 1 s
   "ProdA_SP_Rec2" : Int = PLC ProdA_SP_Rec2 AT %MW200, 1 s
   "ProdA_Tol_Rec2" : Int = PLC ProdA_Tol_Rec2 AT %MW124, 1 s
   "ProdA_SP_Rec3" : Int = PLC ProdA_SP_Rec3 AT %MW138, 1 s
   "ProdA_Tol_Rec3" : Int = PLC ProdA_Tol_Rec3 AT %MW142, 1 s
   "ProdB_SP_Rec1" : Int = PLC ProdB_SP_Rec1 AT %MW102, 1 s
   "ProdB_Tol_Rec1" : Int = PLC ProdB_Tol_Rec1 AT %MW106, 1 s
   "ProdB_SP_Rec2" : Int = PLC ProdB_SP_Rec2 AT %MW122, 1 s
   "ProdB_Tol_Rec2" : Int = PLC ProdB_Tol_Rec2 AT %MW126, 1 s
   "ProdB_SP_Rec3" : Int = PLC ProdB_SP_Rec3 AT %MW140, 1 s
   "ProdB_Tol_Rec3" : Int = PLC ProdB_Tol_Rec3 AT %MW144, 1 s
   "Mix_Temp_SP_Rec1" : Int = PLC Mix_Temp_SP_Rec1 AT %MW108, 1 s
   "Mix_Temp_Tol_Rec1" : Int = PLC Mix_Temp_Tol_Rec1 AT %MW110, 1 s
   "Mix_Temp_SP_Rec2" : Int = PLC Mix_Temp_SP_Rec2 AT %MW128, 1 s
   "Mix_Temp_Tol_Rec2" : Int = PLC Mix_Temp_Tol_Rec2 AT %MW130, 1 s
   "Mix_Temp_SP_Rec3" : Int = PLC Mix_Temp_SP_Rec3 AT %MW146, 1 s
   "Mix_Temp_Tol_Rec3" : Int = PLC Mix_Temp_Tol_Rec3 AT %MW148, 1 s
   "Mix_Time_Rec1" : Int = PLC Mix_Time_Rec1 AT %MW112, 1 s
   "Mix_Time_Rec2" : Int = PLC Mix_Time_Rec2 AT %MW132, 1 s
   "Mix_Time_Rec3" : Int = PLC Mix_Time_Rec3 AT %MW150, 1 s
   "Bottle_Sim_output" : Bool = PLC Bottle_Sim_output AT %Q1.1, 1 s
   "V101_On" : Bool = PLC V101_On AT %Q0.0, 1 s
   "V102_On" : Bool = PLC V102_On AT %Q0.1, 1 s
   "V104_On" : Bool = PLC V104_On AT %Q0.3, 1 s
   "V103_On" : Bool = PLC V103_On AT %Q0.2, 1 s
   "Liquid_Level_Analog" : Int = PLC Liquid_Level_Analog AT %IW66, 1 s
   "Heater_On" : Bool = PLC Heater_On AT %Q0.5, 1 s
   "Mixer_On" : Bool = PLC Mixer_On AT %Q0.4, 1 s
   "Bottle_Count" : Int = PLC Bottle_Count AT %MW156, 1 s
   "Conveyor_On" : Bool = PLC Conveyor_On AT %Q1.0, 1 s
   "V104_Opn" : Bool = PLC V104_Opn AT %I0.6, 1 s
   "V102_Opn" : Bool = PLC V102_Opn AT %I0.2, 1 s
   "V101_Opn" : Bool = PLC V101_Opn AT %I0.0, 1 s
   "V103_Opn" : Bool = PLC V103_Opn AT %I0.4, 1 s
   "V101_Clsd" : Bool = PLC V101_Clsd AT %I0.1, 1 s
   "V102_Clsd" : Bool = PLC V102_Clsd AT %I0.3, 1 s
   "V103_Clsd" : Bool = PLC V103_Clsd AT %I0.5, 1 s
   "V104_Clsd" : Bool = PLC V104_Clsd AT %I0.7, 1 s
   "Reverse_On" : Bool = PLC Reverse_On AT %Q1.1, 1 s
   "Temperature_Measurement_In_PV" : Real = PLC Temperature_Measurement_In.PV, 1 s
   "Conveyor_Speed" : Int = PLC Conveyor_Speed AT %QW80, 1 s
   "Conveyor_Speed_value" : Real = PLC Conveyor_Speed_value AT %MD300, 1 s
   "Mixing_Timer_ET" : Time = PLC Mixing_Timer.ET, 1 s
   "V101_Man" : Bool = PLC V101_Man AT %M165.1, 1 s
   "V102_Man" : Bool = PLC V102_Man AT %M165.2, 1 s
   "V103_Man" : Bool = PLC V103_Man AT %M165.3, 1 s
   "V104_Man" : Bool = PLC V104_Man AT %M165.4, 1 s
   "Heating_Man" : Bool = PLC Heating_Man AT %M165.5, 1 s
   "Conveyor_Man" : Bool = PLC Conveyor_Man AT %M165.6, 1 s
   "Fan_On" : Bool = PLC Fan_On AT %Q0.6, 1 s
   "Bottle_Pos_OK" : Bool = PLC Bottle_Pos_OK AT %I1.2, 1 s
   "Error_Status" : Bool = PLC Error_Status AT %M404.0, 1 s
   "Valve_Error" : Bool = PLC Valve_Error AT %M165.7, 1 s
   "Conveyor_error" : Bool = PLC Conveyor_error AT %M166.1, 1 s
   "Heater_liquid_error" : Bool = PLC Heater_liquid_error AT %M166.0, 1 s
   "Liquid_Error" : Bool = PLC Liquid_Error AT %M166.4, 1 s
   "EMS" : Bool = PLC EMS AT %I1.5, 1 s
   "EMS_Triggered" : Bool = PLC EMS_Triggered AT %M166.6, 1 s

screen "Root screen" 800x480, template "Template_1"
   TextField "HmiScreenItemData_5" at 80,225 size 640x25; Text 'Mixing Tank Simulator'
   Button "HmiScreenItemData_2" at 121,61 size 219x114; TextOff 'Overview Operator Control'; TextOn 'Screen2'; PictureOff "Navigates to Screen2 for KTP700 Basic+ PN 15.0.0.0"; PictureOn "Navigates to Screen2 for KTP700 Basic+ PN 15.0.0.0"
      on Release: ActivateScreen("Overview_Control", 0)
   Button "HmiScreenItemData_3" at 483,61 size 217x115; TextOff 'Manual Control'; TextOn 'Screen3'; PictureOff "Navigates to Screen3 for KTP700 Basic+ PN 15.0.0.0"; PictureOn "Navigates to Screen3 for KTP700 Basic+ PN 15.0.0.0"
      on Release: ActivateScreen("Manual Operation", 0); ResetBit("Manual_Mode")
      on Press: SetBit("Manual_Mode")
   Button "HmiScreenItemData_4" at 196,282 size 409x101; TextOff 'Recipe Management'; TextOn 'Screen4'; PictureOff "Navigates to Screen4 for KTP700 Basic+ PN 15.0.0.0"; PictureOn "Navigates to Screen4 for KTP700 Basic+ PN 15.0.0.0"
      on Release: ActivateScreen("Recipe Management", 0)

screen "Recipe Management" 800x480, template "Template_1"
   Button "Back" at 1,1 size 159x47; TextOff 'Back'
      on Release: ActivateScreen("Root screen", 0)
   TextField "Text field_1" at 332,36 size 75x23; Text 'Recipe 1'
   TextField "Text field_2" at 501,37 size 75x23; Text 'Recipe 2'
   TextField "Text field_3" at 670,37 size 75x23; Text 'Recipe 3'
   TextField "Text field_4" at 10,131 size 267x23; Text 'Product A / Tolerance (+/-) (L):'
   TextField "Text field_6" at 10,63 size 128x23; Text 'Bottle Size (L):'
   TextField "Text field_7" at 10,96 size 117x23; Text 'No of Bottles:'
   TextField "Text field_5" at 10,165 size 266x23; Text 'Product B / Tolerance (+/-) (L):'
   TextField "Text field_8" at 10,200 size 269x23; Text 'Mix Temp / Tolerance (+/-) (C):'
   TextField "Text field_9" at 9,237 size 130x23; Text 'Mix Time (mS):'
   IOField "I/O field_1" at 340,63 size 53x27; FormatPattern s99999
      ProcessValue <- "Bottle_Size_Rec1"
   IOField "I/O field_2" at 680,69 size 53x27; FormatPattern s99999
      ProcessValue <- "Bottle_Size_Rec3"
   IOField "I/O field_3" at 510,69 size 53x27; FormatPattern s99999
      ProcessValue <- "Bottle_Size_Rec2"
   IOField "I/O field_4" at 340,90 size 53x27; FormatPattern s99999
      ProcessValue <- "Bottle_Batch_Size_Rec1"
   IOField "I/O field_5" at 510,92 size 53x27; FormatPattern s99999
      ProcessValue <- "Bottle_Batch_Size_Rec2"
   IOField "I/O field_6" at 680,98 size 53x27; FormatPattern s99999
      ProcessValue <- "Bottle_Batch_Size_Rec3"
   IOField "I/O field_7" at 312,133 size 52x27; FormatPattern s99999
      ProcessValue <- "ProdA_SP_Rec1"
   IOField "I/O field_8" at 365,133 size 52x27; FormatPattern s99999
      ProcessValue <- "ProdA_Tol_Rec1"
   IOField "I/O field_9" at 483,133 size 52x27; FormatPattern s99999
      ProcessValue <- "ProdA_SP_Rec2"
   IOField "I/O field_10" at 536,133 size 52x27; FormatPattern s99999
      ProcessValue <- "ProdA_Tol_Rec2"
   IOField "I/O field_11" at 655,133 size 52x27; FormatPattern s99999
      ProcessValue <- "ProdA_SP_Rec3"
   IOField "I/O field_12" at 708,133 size 52x27; FormatPattern s99999
      ProcessValue <- "ProdA_Tol_Rec3"
   IOField "I/O field_13" at 312,161 size 52x27; FormatPattern s99999
      ProcessValue <- "ProdB_SP_Rec1"
   IOField "I/O field_14" at 365,161 size 52x27; FormatPattern s99999
      ProcessValue <- "ProdB_Tol_Rec1"
   IOField "I/O field_15" at 483,160 size 52x27; FormatPattern s99999
      ProcessValue <- "ProdB_SP_Rec2"
   IOField "I/O field_16" at 536,160 size 52x27; FormatPattern s99999
      ProcessValue <- "ProdB_Tol_Rec2"
   IOField "I/O field_17" at 655,159 size 52x27; FormatPattern s99999
      ProcessValue <- "ProdB_SP_Rec3"
   IOField "I/O field_18" at 708,159 size 52x27; FormatPattern s99999
      ProcessValue <- "ProdB_Tol_Rec3"
   IOField "I/O field_19" at 312,200 size 52x27; FormatPattern s99999
      ProcessValue <- "Mix_Temp_SP_Rec1"
   IOField "I/O field_20" at 365,200 size 52x27; FormatPattern s99999
      ProcessValue <- "Mix_Temp_Tol_Rec1"
   IOField "I/O field_21" at 314,236 size 104x27; FormatPattern 99999
      ProcessValue <- "Mix_Time_Rec1"
   IOField "I/O field_23" at 483,196 size 52x27; FormatPattern s99999
      ProcessValue <- "Mix_Temp_SP_Rec2"
   IOField "I/O field_24" at 536,196 size 52x27; FormatPattern s99999
      ProcessValue <- "Mix_Temp_Tol_Rec2"
   IOField "I/O field_25" at 655,196 size 52x27; FormatPattern s99999
      ProcessValue <- "Mix_Temp_SP_Rec3"
   IOField "I/O field_26" at 708,196 size 52x27; FormatPattern s99999
      ProcessValue <- "Mix_Temp_Tol_Rec3"
   IOField "I/O field_28" at 656,237 size 102x27; FormatPattern 99999
      ProcessValue <- "Mix_Time_Rec3"
   IOField "I/O field_30" at 484,236 size 103x27; FormatPattern 99999
      ProcessValue <- "Mix_Time_Rec2"

screen "Manual Operation" 800x480, template "Template_1"
   TextField "HmiScreenItemData" at 127,3 size 640x25; Text 'Manual Process Operation'
   Button "Back" at 1,1 size 159x47; TextOn 'Back'; TextOff 'Back'
      on Release: ActivateScreen("Root screen", 0)
   Button "Button_4" at 627,85 size 168x64; TextOff 'Recipe 1'
      on Release: ResetBit("Recipe_1")
      on Press: SetBit("Recipe_1")
   Button "Button_5" at 628,157 size 168x64; TextOff 'Recipe 2'
      on Release: ResetBit("Recipe_2")
      on Press: SetBit("Recipe_2")
   Button "Button_6" at 628,229 size 168x64; TextOff 'Recipe 3'
      on Release: ResetBit("Recipe_3")
      on Press: SetBit("Recipe_3")
   Switch "Switch_1" at 17,78 size 162x55; TextOn 'ON'; CaptionText 'Switch'; TextOff 'OFF'
      ProcessValue <- "V101_Man"
   TextField "Text field_1" at 195,94 size 127x29; Text 'Valve V101'
   Switch "Switch_2" at 18,140 size 162x55; TextOn 'ON'; CaptionText 'Switch'; TextOff 'OFF'
      ProcessValue <- "V102_Man"
   TextField "Text field_2" at 196,156 size 127x29; Text 'Valve V102'
   Switch "Switch_3" at 19,202 size 162x55; TextOn 'ON'; CaptionText 'Switch'; TextOff 'OFF'
      ProcessValue <- "V103_Man"
   TextField "Text field_3" at 197,218 size 127x29; Text 'Valve V103'
   Switch "Switch_4" at 20,264 size 162x55; TextOn 'ON'; CaptionText 'Switch'; TextOff 'OFF'
      ProcessValue <- "V104_Man"
   TextField "Text field_4" at 198,280 size 127x29; Text 'Valve V104'
   Circle "Circle_1" at 326,86 size 39x39
      Appearance <- "V101_On"
   Circle "Circle_2" at 326,152 size 39x39
      Appearance <- "V102_On"
   Circle "Circle_3" at 326,214 size 39x39
      Appearance <- "V103_On"
   Circle "Circle_4" at 326,274 size 39x39
      Appearance <- "V104_On"
   TextField "Text field_5" at 329,48 size 27x23; Text 'On'
   TextField "Text field_6" at 395,48 size 47x23; Text 'Open'
   TextField "Text field_7" at 461,48 size 59x23; Text 'Closed'
   TextField "Text field_8" at 535,48 size 94x23; Text 'Tank Level'
   Switch "Switch_5" at 20,327 size 162x55; TextOn 'ON'; CaptionText 'Switch'; TextOff 'OFF'
      ProcessValue <- "Conveyor_Man"
   TextField "Text field_9" at 186,339 size 138x29; Text 'Conveyor On'
   Circle "Circle_5" at 326,337 size 39x39
      Appearance <- "Conveyor_On"
   Circle "Circle_6" at 401,86 size 39x39
      Appearance <- "V101_Opn"
   Circle "Circle_7" at 401,152 size 39x39
      Appearance <- "V102_Opn"
   Circle "Circle_8" at 401,214 size 39x39
      Appearance <- "V103_Opn"
   Circle "Circle_9" at 401,274 size 39x39
      Appearance <- "V104_Opn"
   Circle "Circle_10" at 476,86 size 39x39
      Appearance <- "V101_Clsd"
   Circle "Circle_11" at 476,152 size 39x39
      Appearance <- "V102_Clsd"
   Circle "Circle_12" at 476,214 size 39x39
      Appearance <- "V103_Clsd"
   Circle "Circle_13" at 476,274 size 39x39
      Appearance <- "V104_Clsd"
   TextField "Text field_10" at 643,48 size 140x23; Text 'Recipe Selection'
   Button "Button_9" at 628,300 size 95x68; TextOff 'Bottle'
      on Release: ResetBit("Bottle_Sim_output")
      on Press: SetBit("Bottle_Sim_output")
   Circle "Circle_14" at 734,309 size 53x53
      Appearance <- "Bottle_Pos_OK"
   Switch "Switch_6" at 20,384 size 162x27; TextOn 'Reverse'; CaptionText 'Switch'; TextOff 'Forward'
      ProcessValue <- "Reverse_On"
   TextField "Text field_11" at 377,340 size 88x29; Text 'Reverse'
   Circle "Circle_15" at 476,337 size 39x39
      Appearance <- "Reverse_On"
   Button "Button_2" at 182,3 size 133x46; TextOff 'Reset'
      on Release: ResetBit("Reset_PB")
      on Press: SetBit("Reset_PB")
   Switch "Switch_7" at 20,414 size 162x28; TextOn 'ON'; CaptionText 'Switch'; TextOff 'OFF'
      ProcessValue <- "Heating_Man"
   TextField "Text field_12" at 186,413 size 111x29; Text 'Heater On'
   Circle "Circle_16" at 300,414 size 28x28
      Appearance <- "Heater_On"
   IOField "I/O field_1" at 696,2 size 86x25; FormatPattern s99999
      ProcessValue <- "Bottle_Count"
   TextField "Text field_13" at 583,1 size 108x23; Text 'Bottle Count'
   IOField "I/O field_2" at 696,27 size 86x25; FormatPattern 99.99
      ProcessValue <- "Temperature_Measurement_In_PV"
   TextField "Text field_14" at 583,24 size 81x23; Text 'Temp (C)'
   Switch "Switch_8" at 437,415 size 162x55; TextOn 'ON'; CaptionText 'Switch'; TextOff 'OFF'
      ProcessValue <- "Mixer_On"
   TextField "Text field_15" at 613,427 size 99x29; Text 'Mixer On'
   Circle "Circle_17" at 743,425 size 39x39
      Appearance <- "Mixer_On"
   IOField "I/O field_3" at 332,383 size 53x31; FormatPattern 99999
      ProcessValue <- "Conveyor_Speed_value"
   TextField "Text field_16" at 187,386 size 136x23; Text 'Conveyor Speed'
   Bar "Bar_2" at 544,79 size 69x303; MinimumValue 0; MaximumValue 100
      ProcessValue <- "TankSimulator_DB_Level"
   Switch "Switch_9" at 20,442 size 162x28; TextOn 'ON'; CaptionText 'Switch'; TextOff 'OFF'
      ProcessValue <- "Fan_On"
   TextField "Text field_17" at 187,441 size 78x29; Text 'Fan On'
   Circle "Circle_18" at 300,444 size 28x28
      Appearance <- "Fan_On"

screen "Overview_Control" 800x480, template "Template_1"
   Button "Back" at 1,1 size 159x47; TextOn 'Back'; TextOff 'Back'
      on Release: ActivateScreen("Root screen", 0)
   GraphicView "Graphic view_1" at 245,95 size 177x231; Picture "Graphic_1"
   GraphicView "Graphic view_2" at 401,14 size 67x78; Picture "Graphic_2"
   GraphicView "Graphic view_3" at 209,14 size 67x78; Picture "Graphic_2"
   GraphicView "Graphic view_4" at 416,296 size 65x72; Picture "Graphic_2"
   GraphicView "Graphic view_6" at 109,291 size 67x78; Picture "Graphic_2"
   GraphicView "Graphic view_7" at 306,319 size 52x43; Picture "Graphic_3"
   GraphicView "Graphic view_8" at 355,333 size 66x35; Picture "Graphic_4"
   GraphicView "Graphic view_9" at 475,342 size 37x36; Picture "Graphic_5"
   GraphicView "Graphic view_10" at 172,332 size 140x38; Picture "Graphic_6"
   GraphicView "Graphic view_11" at 62,336 size 50x46; Picture "Graphic_7"
   GraphicView "Graphic view_12" at 358,60 size 46x48; Picture "Graphic_7"
   GraphicView "Graphic view_13" at 274,60 size 48x48; Picture "Graphic_5"
   GraphicView "Graphic view_14" at 462,57 size 103x30; Picture "Graphic_4"
   GraphicView "Graphic view_15" at 110,58 size 103x30; Picture "Graphic_4"
   Bar "Bar_1" at 318,124 size 69x174; MinimumValue 0; MaximumValue 1000
      ProcessValue <- "TankSimulator_DB_Level"
   TextField "Text field_1" at 167,13 size 46x23; Text 'V101'
   TextField "Text field_2" at 358,14 size 46x23; Text 'V102'
   TextField "Text field_3" at 481,307 size 46x23; Text 'V103'
   TextField "Text field_4" at 63,291 size 46x23; Text 'V104'
   GraphicView "Graphic view_5" at 263,400 size 357x69; Picture "Graphic_8"
   GraphicView "Graphic view_16" at 378,122 size 90x167; Picture "Graphic_9"
   TextField "Text field_5" at 429,108 size 51x23; Text 'Mixer'
   GraphicView "Graphic view_17" at 249,238 size 42x64; Picture "Graphic_11"
   TextField "Text field_6" at 188,226 size 61x23; Text 'Heater'
   GraphicView "Graphic view_18" at 481,382 size 50x52; Picture "Graphic_12"
   GraphicView "Graphic view_19" at 418,383 size 50x52; Picture "Graphic_12"
   GraphicView "Graphic view_20" at 355,384 size 50x52; Picture "Graphic_12"
   Rectangle "Rectangle_3" at 419,19 size 31x16
      Visibility <- "V102_On"
   Rectangle "Rectangle_5" at 126,296 size 31x16
      Visibility <- "V104_On"
   Rectangle "Rectangle_7" at 433,300 size 31x16
      Visibility <- "V103_On"
   Rectangle "Rectangle_10" at 455,173 size 31x16
      Visibility <- "Mixer_On"
   Rectangle "Rectangle_9" at 273,220 size 31x16
      Visibility <- "Heater_On"
   Button "Button_1" at 627,8 size 168x64; TextOff 'Start'
      on Release: ResetBit("Start_PB")
      on Press: SetBit("Start_PB")
   Button "Button_7" at 627,81 size 168x64; TextOff 'Automatic'
      on Press: SetBit("Auto_Mode")
      on Release: ResetBit("Auto_Mode")
   Button "Button_4" at 627,152 size 168x64; TextOff 'Recipe 1'
      on Release: ResetBit("Recipe_1")
      on Press: SetBit("Recipe_1")
   Button "Button_5" at 628,224 size 168x64; TextOff 'Recipe 2'
      on Release: ResetBit("Recipe_2")
      on Press: SetBit("Recipe_2")
   Button "Button_6" at 628,296 size 168x64; TextOff 'Recipe 3'
      on Release: ResetBit("Recipe_3")
      on Press: SetBit("Recipe_3")
   IOField "I/O field_1" at 263,409 size 86x25; FormatPattern s99999
      ProcessValue <- "Bottle_Count"
   TextField "Text field_7" at 150,408 size 108x23; Text 'Bottle Count'
   Rectangle "Rectangle_2" at 301,443 size 31x16
      Visibility <- "Conveyor_On"
   Rectangle "Rectangle_4" at 356,443 size 31x16
      Visibility <- "Conveyor_On"
   Rectangle "Rectangle_6" at 414,443 size 31x16
      Visibility <- "Conveyor_On"
   Rectangle "Rectangle_8" at 470,443 size 31x16
      Visibility <- "Conveyor_On"
   Rectangle "Rectangle_11" at 528,443 size 31x16
      Visibility <- "Conveyor_On"
   Button "Button_2" at 13,199 size 168x64; TextOff 'Reset'
      on Release: ResetBit("Reset_PB")
      on Press: SetBit("Reset_PB")
   IOField "I/O field_2" at 192,248 size 54x25; FormatPattern 99.99
      ProcessValue <- "Temperature_Measurement_In_PV"
   Button "Button_3" at 13,130 size 168x64; TextOff 'Stop'
      on Release: ResetBit("Stop_PB")
      on Press: SetBit("Stop_PB")
   Button "Button_9" at 629,371 size 168x64; TextOff 'Bottle Presence'
      on Release: ResetBit("Bottle_Sim_output")
      on Press: SetBit("Bottle_Sim_output")
   IOField "I/O field_3" at 172,437 size 86x25; FormatPattern 99999
      ProcessValue <- "Conveyor_Speed_value"
   TextField "Text field_8" at 28,437 size 136x23; Text 'Conveyor Speed'
   Bar "Bar_2" at 318,124 size 69x174; MinimumValue 0; MaximumValue 100
      ProcessValue <- "TankSimulator_DB_Level"
   Rectangle "Rectangle_1" at 227,19 size 31x16
      Visibility <- "V101_On"
   IOField "I/O field_4" at 192,187 size 54x25; FormatPattern s9999999999
      ProcessValue <- "Mixing_Timer_ET"
   TextField "Text field_9" at 192,163 size 53x23; Text 'Timer'
   Circle "Circle_1" at 581,209 size 24x24
      Appearance <- "Valve_Error"
   TextField "Text field_10" at 473,210 size 50x23; Text 'Valve'
   Circle "Circle_2" at 581,236 size 24x24
      Appearance <- "Conveyor_error"
   TextField "Text field_11" at 472,236 size 81x23; Text 'Conveyor'
   Circle "Circle_3" at 581,262 size 24x24
      Appearance <- "Liquid_Error"
   TextField "Text field_12" at 466,266 size 107x23; Text 'Liquid Level'
   TextField "Text field_13" at 512,148 size 54x23; Text 'Errors'
   Circle "Circle_4" at 581,180 size 24x24
      Appearance <- "EMS_Triggered"
   TextField "Text field_14" at 492,181 size 39x23; Text 'EMS'
*)

(* ===== HMI "HMI_RT_2" =====
system functions are stored by id; their names below are inferred from use
connection "HMI_Connection_3": ETHERNET, S7_1200_OMS
connection "HMI_Connection_4": ETHERNET, S7_1200_OMS

HMI tags "Default tag table"
   "Stop_PB" : Bool = PLC Stop_PB AT %M11.0, 1 s
   "Reset_PB" : Bool = PLC Reset_PB AT %M15.0, 1 s
   "V101_On" : Bool = PLC V101_On AT %Q0.0, 1 s
   "V102_On" : Bool = PLC V102_On AT %Q0.1, 1 s
   "Mixer_On" : Bool = PLC Mixer_On AT %Q0.4, 1 s
   "Heater_On" : Bool = PLC Heater_On AT %Q0.5, 1 s
   "V103_On" : Bool = PLC V103_On AT %Q0.2, 1 s
   "V104_On" : Bool = PLC V104_On AT %Q0.3, 1 s
   "Start_PB" : Bool = PLC Start_PB AT %M10.0, 1 s
   "Auto_Mode" : Bool = PLC Auto_Mode AT %M12.0, 1 s
   "Recipe_1" : Bool = PLC Recipe_1 AT %M118.0, 1 s
   "Recipe_2" : Bool = PLC Recipe_2 AT %M119.0, 1 s
   "Recipe_3" : Bool = PLC Recipe_3 AT %M120.0, 1 s
   "Bottle_Sim_output" : Bool = PLC Bottle_Sim_output AT %Q1.1, 1 s
   "Conveyor_On" : Bool = PLC Conveyor_On AT %Q1.0, 1 s
   "Conveyor_Speed_value" : Real = PLC Conveyor_Speed_value AT %MD300, 1 s
   "Bottle_Count" : Int = PLC Bottle_Count AT %MW156, 1 s
   "Recipe Selection_DB_Bottle_Size" : Int = PLC "Recipe Selection_DB".Bottle_Size, 1 s
   "Recipe Selection_DB_Bottle_Number" : Int = PLC "Recipe Selection_DB".Bottle_Number, 1 s
   "Recipe Selection_DB_Product_A" : Int = PLC "Recipe Selection_DB".Product_A, 1 s
   "Recipe Selection_DB_Product_B" : Int = PLC "Recipe Selection_DB".Product_B, 1 s
   "Recipe Selection_DB_Mix_Temp" : Int = PLC "Recipe Selection_DB".Mix_Temp, 1 s
   "Recipe Selection_DB_Mixing_Time" : DInt = PLC "Recipe Selection_DB".Mixing_Time, 1 s
   "Bottle_Pos_OK" : Bool = PLC Bottle_Pos_OK AT %I1.2, 1 s
   "Temperature_Measurement_In_PV" : Real = PLC Temperature_Measurement_In.PV, 1 s
   "Liquid_Level_Analog" : Int = PLC Liquid_Level_Analog AT %IW66, 1 s
   "Mixing_Timer_ET" : Time = PLC Mixing_Timer.ET, 1 s
   "End_cycle" : Bool = PLC End_cycle AT %M165.0, 1 s
   "Step_2" : Bool = PLC Step_2 AT %M51.0, 1 s
   "Step_3" : Bool = PLC Step_3 AT %M52.0, 1 s
   "Step_4" : Bool = PLC Step_4 AT %M53.0, 1 s
   "Step_5" : Bool = PLC Step_5 AT %M54.0, 1 s
   "Step_6" : Bool = PLC Step_6 AT %M55.0, 1 s
   "Step_7" : Bool = PLC Step_7 AT %M56.0, 1 s
   "Step_8" : Bool = PLC Step_8 AT %M60.0, 1 s
   "Step_9" : Bool = PLC Step_9 AT %M58.0, 1 s
   "Bottle_Size_Rec1" : Int = PLC Bottle_Size_Rec1 AT %MW114, 1 s
   "Bottle_Size_Rec2" : Int = PLC Bottle_Size_Rec2 AT %MW134, 1 s
   "Bottle_Size_Rec3" : Int = PLC Bottle_Size_Rec3 AT %MW152, 1 s
   "Bottle_Batch_Size_Rec1" : Int = PLC Bottle_Batch_Size_Rec1 AT %MW116, 1 s
   "Bottle_Batch_Size_Rec2" : Int = PLC Bottle_Batch_Size_Rec2 AT %MW136, 1 s
   "Bottle_Batch_Size_Rec3" : Int = PLC Bottle_Batch_Size_Rec3 AT %MW154, 1 s
   "ProdA_SP_Rec1" : Int = PLC ProdA_SP_Rec1 AT %MW100, 1 s
   "ProdA_Tol_Rec1" : Int = PLC ProdA_Tol_Rec1 AT %MW104, 1 s
   "ProdA_SP_Rec2" : Int = PLC ProdA_SP_Rec2 AT %MW200, 1 s
   "ProdA_Tol_Rec2" : Int = PLC ProdA_Tol_Rec2 AT %MW124, 1 s
   "ProdA_SP_Rec3" : Int = PLC ProdA_SP_Rec3 AT %MW138, 1 s
   "ProdA_Tol_Rec3" : Int = PLC ProdA_Tol_Rec3 AT %MW142, 1 s
   "ProdB_SP_Rec1" : Int = PLC ProdB_SP_Rec1 AT %MW102, 1 s
   "ProdB_SP_Rec2" : Int = PLC ProdB_SP_Rec2 AT %MW122, 1 s
   "ProdB_SP_Rec3" : Int = PLC ProdB_SP_Rec3 AT %MW140, 1 s
   "ProdB_Tol_Rec3" : Int = PLC ProdB_Tol_Rec3 AT %MW144, 1 s
   "ProdB_Tol_Rec2" : Int = PLC ProdB_Tol_Rec2 AT %MW126, 1 s
   "ProdB_Tol_Rec1" : Int = PLC ProdB_Tol_Rec1 AT %MW106, 1 s
   "Mix_Temp_SP_Rec1" : Int = PLC Mix_Temp_SP_Rec1 AT %MW108, 1 s
   "Mix_Temp_SP_Rec2" : Int = PLC Mix_Temp_SP_Rec2 AT %MW128, 1 s
   "Mix_Temp_SP_Rec3" : Int = PLC Mix_Temp_SP_Rec3 AT %MW146, 1 s
   "Mix_Temp_Tol_Rec3" : Int = PLC Mix_Temp_Tol_Rec3 AT %MW148, 1 s
   "Mix_Temp_Tol_Rec2" : Int = PLC Mix_Temp_Tol_Rec2 AT %MW130, 1 s
   "Mix_Temp_Tol_Rec1" : Int = PLC Mix_Temp_Tol_Rec1 AT %MW110, 1 s
   "Mix_Time_Rec1" : Int = PLC Mix_Time_Rec1 AT %MW112, 1 s
   "Mix_Time_Rec2" : Int = PLC Mix_Time_Rec2 AT %MW132, 1 s
   "Mix_Time_Rec3" : Int = PLC Mix_Time_Rec3 AT %MW150, 1 s
   "Step_1" : Bool = PLC Step_1 AT %M50.0, 1 s
   "Ultrasonic_Lvl_In_DB_PV" : Real = PLC Ultrasonic_Lvl_In_DB.PV, 1 s
   "ProdA_Level_Error" : Bool = PLC ProdA_Level_Error AT %M166.2, 1 s
   "ProdB_Level_Error" : Bool = PLC ProdB_Level_Error AT %M166.3, 1 s
   "Heater_liquid_error" : Bool = PLC Heater_liquid_error AT %M166.0, 1 s
   "Conveyor_error" : Bool = PLC Conveyor_error AT %M166.1, 1 s
   "Overflow_Error" : Bool = PLC Overflow_Error AT %M166.5, 1 s
   "EMS_Triggered" : Bool = PLC EMS_Triggered AT %M166.6, 1 s

